C03641=1085.431,193.787,426.728,175.436,21.892,153.539
C03642=1085.437,194.036,426.705,175.438,21.893,153.539
C03643=1085.443,194.285,426.682,175.441,21.895,153.539
C03644=1085.448,194.534,426.658,175.443,21.897,153.539
C03645=1085.453,194.783,426.636,175.446,21.899,153.539
C03646=1085.459,195.032,426.613,175.448,21.900,153.539
C03647=1085.465,195.280,426.589,175.451,21.902,153.539
C03648=1085.470,195.530,426.565,175.453,21.904,153.539
C03649=1085.476,195.779,426.542,175.457,21.906,153.539
C03650=1085.482,196.027,426.519,175.459,21.907,153.539
C03651=1085.487,196.277,426.496,175.461,21.909,153.539
C03652=1085.493,196.525,426.472,175.464,21.911,153.539
C03653=1085.498,196.774,426.449,175.467,21.912,153.539
C03654=1085.504,197.023,426.426,175.469,21.914,153.539
C03655=1085.510,197.271,426.402,175.471,21.916,153.539
C03656=1085.515,197.520,426.379,175.474,21.917,153.539
C03657=1085.521,197.769,426.356,175.476,21.919,153.539
C03658=1085.526,198.018,426.333,175.479,21.921,153.539
C03659=1085.532,198.267,426.309,175.482,21.923,153.539
C03660=1085.538,198.515,426.286,175.485,21.925,153.539
C03661=1085.543,198.765,426.263,175.487,21.927,153.539
C03662=1085.549,199.013,426.239,175.490,21.928,153.539
C03663=1085.554,199.262,426.216,175.492,21.930,153.539
C03664=1085.560,199.510,426.192,175.495,21.932,153.539
C03665=1085.566,199.759,426.169,175.497,21.933,153.539
C03666=1085.572,200.009,426.145,175.500,21.935,153.539
C03667=1085.577,200.258,426.121,175.502,21.937,153.539
C03668=1085.583,200.506,426.098,175.505,21.938,153.539
C03669=1085.589,200.755,426.075,175.508,21.940,153.539
C03670=1085.594,201.004,426.051,175.511,21.942,153.538
C03671=1085.600,201.252,426.027,175.513,21.944,153.539
C03672=1085.605,201.501,426.004,175.516,21.945,153.539
C03673=1085.612,201.750,425.980,175.518,21.947,153.538
C03674=1085.617,201.999,425.957,175.521,21.949,153.538
C03675=1085.623,202.248,425.933,175.523,21.950,153.538
C03676=1085.628,202.497,425.910,175.526,21.952,153.538
C03677=1085.634,202.745,425.885,175.529,21.954,153.538
C03678=1085.639,202.994,425.862,175.532,21.956,153.538
C03679=1085.645,203.243,425.838,175.534,21.957,153.538
C03680=1085.651,203.492,425.815,175.537,21.959,153.538
C03681=1085.656,203.741,425.791,175.539,21.961,153.538
C03682=1085.661,203.990,425.767,175.542,21.963,153.538
C03683=1085.667,204.239,425.743,175.544,21.964,153.538
C03684=1085.673,204.487,425.719,175.548,21.966,153.538
C03685=1085.678,204.736,425.696,175.550,21.968,153.538
C03686=1085.684,204.985,425.672,175.553,21.970,153.538
C03687=1085.689,205.233,425.648,175.555,21.972,153.538
C03688=1085.695,205.483,425.624,175.558,21.973,153.538
C03689=1085.701,205.731,425.600,175.560,21.975,153.538
C03690=1085.706,205.980,425.576,175.564,21.977,153.538
C03691=1085.712,206.229,425.553,175.566,21.979,153.538
C03692=1085.717,206.477,425.529,175.568,21.981,153.538
C03693=1085.724,206.726,425.505,175.571,21.983,153.538
C03694=1085.729,206.976,425.481,175.574,21.984,153.538
C03695=1085.734,207.224,425.457,175.576,21.986,153.538
C03696=1085.757,208.251,425.358,175.658,22.028,153.535
C03697=1085.767,208.639,425.320,175.662,22.033,153.535
C03698=1085.775,209.027,425.282,175.666,22.037,153.535
C03699=1085.783,209.415,425.244,175.670,22.041,153.536
C03700=1085.793,209.803,425.205,175.673,22.045,153.536
C03701=1085.798,210.051,425.181,175.676,22.048,153.536
C03702=1085.804,210.301,425.157,175.678,22.050,153.536
C03703=1085.810,210.549,425.132,175.681,22.053,153.536
C03704=1085.815,210.798,425.108,175.684,22.056,153.537
C03705=1085.821,211.047,425.083,175.686,22.058,153.537
C03706=1085.826,211.295,425.058,175.689,22.061,153.537
C03707=1085.832,211.544,425.034,175.691,22.064,153.537
C03708=1085.838,211.793,425.010,175.694,22.067,153.538
C03709=1085.843,212.042,424.985,175.696,22.069,153.538
C03710=1085.849,212.290,424.960,175.699,22.072,153.538
C03711=1085.854,212.539,424.936,175.701,22.075,153.538
C03712=1085.860,212.788,424.911,175.704,22.077,153.538
C03713=1085.866,213.036,424.886,175.707,22.080,153.538
C03714=1085.872,213.285,424.862,175.709,22.083,153.539
C03715=1085.877,213.534,424.837,175.712,22.086,153.539
C03716=1085.882,213.784,424.812,175.714,22.088,153.539
C03717=1085.888,214.032,424.787,175.716,22.091,153.539
C03718=1085.894,214.281,424.762,175.720,22.094,153.539
C03719=1085.899,214.529,424.737,175.722,22.096,153.540
C03720=1085.905,214.777,424.713,175.725,22.099,153.540
C03721=1085.910,215.027,424.689,175.727,22.102,153.540
C03722=1085.916,215.275,424.664,175.730,22.105,153.540
C03723=1085.921,215.524,424.638,175.732,22.107,153.540
C03724=1085.927,215.772,424.613,175.734,22.110,153.541
C03725=1085.933,216.022,424.589,175.737,22.113,153.541
C03726=1085.938,216.270,424.564,175.740,22.115,153.541
C03727=1085.944,216.519,424.539,175.743,22.118,153.541
C03728=1085.949,216.767,424.514,175.745,22.121,153.541
C03729=1085.955,217.016,424.489,175.748,22.124,153.542
C03730=1085.961,217.264,424.464,175.750,22.126,153.542
C03731=1085.967,217.514,424.439,175.753,22.129,153.542
C03732=1085.973,217.762,424.414,175.755,22.132,153.542
C03733=1085.977,218.011,424.389,175.757,22.134,153.542
C03734=1085.984,218.260,424.364,175.761,22.137,153.543
C03735=1085.989,218.508,424.340,175.763,22.139,153.543
C03736=1085.995,218.757,424.314,175.766,22.143,153.543
C03737=1086.000,219.006,424.290,175.768,22.145,153.543
C03738=1086.006,219.255,424.264,175.771,22.148,153.543
C03739=1086.012,219.503,424.239,175.773,22.151,153.544
C03740=1086.017,219.752,424.215,175.776,22.153,153.544
C03741=1086.023,220.001,424.189,175.779,22.156,153.544
C03742=1086.028,220.249,424.164,175.782,22.159,153.544
C03743=1086.034,220.498,424.139,175.784,22.161,153.544
C03744=1086.040,220.747,424.114,175.786,22.164,153.544
C03745=1086.046,220.995,424.089,175.789,22.167,153.545
C03746=1086.051,221.244,424.063,175.791,22.169,153.545
C03747=1086.057,221.493,424.038,175.794,22.172,153.545
C03748=1086.063,221.741,424.013,175.797,22.175,153.545
C03749=1086.072,222.133,423.973,175.801,22.179,153.546
C03750=1086.081,222.526,423.934,175.805,22.183,153.546
C03751=1086.090,222.917,423.893,175.809,22.188,153.546
C03752=1086.098,223.309,423.854,175.813,22.192,153.547
C03753=1086.103,223.558,423.828,175.816,22.195,153.547
C03754=1086.109,223.806,423.803,175.818,22.197,153.547
C03755=1086.115,224.054,423.778,175.821,22.201,153.547
C03756=1086.121,224.303,423.752,175.824,22.203,153.547
C03757=1086.126,224.553,423.727,175.827,22.206,153.548
C03758=1086.131,224.801,423.702,175.829,22.209,153.548
C03759=1086.138,225.050,423.676,175.832,22.211,153.548
C03760=1086.143,225.298,423.650,175.834,22.214,153.548
C03761=1086.149,225.546,423.625,175.837,22.217,153.548
C03762=1086.154,225.795,423.599,175.839,22.219,153.548
C03763=1086.160,226.044,423.574,175.842,22.223,153.549
C03764=1086.165,226.292,423.548,175.845,22.225,153.549
C03765=1086.171,226.541,423.523,175.848,22.228,153.549
C03766=1086.177,226.790,423.497,175.850,22.231,153.549
C03767=1086.182,227.039,423.471,175.853,22.233,153.549
C03768=1086.188,227.287,423.446,175.855,22.236,153.550
C03769=1086.193,227.536,423.420,175.858,22.239,153.550
C03770=1086.200,227.785,423.395,175.860,22.241,153.550
C03771=1086.205,228.034,423.369,175.863,22.245,153.550
C03772=1086.211,228.282,423.344,175.866,22.247,153.551
C03773=1086.216,228.531,423.318,175.869,22.250,153.551
C03774=1086.222,228.779,423.293,175.871,22.252,153.551
C03775=1086.228,229.028,423.267,175.874,22.255,153.551
C03776=1086.234,229.277,423.240,175.876,22.258,153.551
C03777=1086.239,229.525,423.215,175.879,22.261,153.552
C03778=1086.245,229.774,423.189,175.881,22.263,153.552
C03779=1086.251,230.022,423.164,175.885,22.266,153.552
C03780=1086.256,230.271,423.138,175.887,22.269,153.552
C03781=1086.262,230.520,423.112,175.890,22.272,153.552
C03782=1086.267,230.768,423.087,175.892,22.274,153.552
C03783=1086.273,231.016,423.061,175.895,22.277,153.553
C03784=1086.279,231.265,423.035,175.898,22.280,153.553
C03785=1086.284,231.514,423.009,175.900,22.283,153.553
C03786=1086.290,231.763,422.983,175.903,22.285,153.553
C03787=1086.295,232.011,422.957,175.905,22.288,153.554
C03788=1086.301,232.260,422.931,175.909,22.291,153.554
C03789=1086.306,232.509,422.905,175.911,22.293,153.554
C03790=1086.313,232.757,422.880,175.914,22.297,153.554
C03791=1086.318,233.006,422.853,175.916,22.299,153.554
C03792=1086.324,233.255,422.827,175.919,22.302,153.555
C03793=1086.329,233.503,422.802,175.921,22.305,153.555
C03794=1086.335,233.751,422.776,175.924,22.307,153.555
C03795=1086.341,234.000,422.750,175.927,22.310,153.555
C03796=1086.346,234.248,422.723,175.930,22.313,153.555
C03797=1086.352,234.497,422.697,175.933,22.316,153.556
C03798=1086.357,234.746,422.671,175.935,22.319,153.556
C03799=1086.363,234.995,422.645,175.938,22.322,153.556
C03800=1086.368,235.243,422.619,175.940,22.324,153.556
C03801=1086.377,235.626,422.579,175.945,22.329,153.556
C03802=1086.386,236.010,422.538,175.948,22.333,153.557
C03803=1086.394,236.393,422.498,175.953,22.337,153.557
C03804=1086.404,236.777,422.458,175.957,22.341,153.557
C03805=1086.409,237.025,422.431,175.960,22.344,153.558
C03806=1086.414,237.273,422.405,175.962,22.347,153.558
C03807=1086.420,237.522,422.379,175.965,22.350,153.558
C03808=1086.425,237.771,422.353,175.968,22.353,153.558
C03809=1086.431,238.019,422.326,175.970,22.355,153.558
C03810=1086.437,238.267,422.300,175.973,22.359,153.559
C03811=1086.442,238.516,422.274,175.976,22.361,153.559
C03812=1086.448,238.765,422.247,175.979,22.364,153.559
C03813=1086.454,239.014,422.221,175.981,22.366,153.559
C03814=1086.459,239.262,422.194,175.984,22.369,153.559
C03815=1086.465,239.510,422.168,175.987,22.372,153.560
C03816=1086.471,239.759,422.142,175.989,22.375,153.560
C03817=1086.476,240.008,422.115,175.992,22.378,153.560
C03818=1086.482,240.256,422.088,175.994,22.380,153.560
C03819=1086.488,240.505,422.063,175.998,22.383,153.560
C03820=1086.493,240.753,422.036,176.001,22.386,153.561
C03821=1086.499,241.002,422.009,176.003,22.389,153.561
C03822=1086.505,241.250,421.983,176.006,22.391,153.561
C03823=1086.510,241.499,421.957,176.008,22.394,153.561
C03824=1086.516,241.747,421.930,176.011,22.397,153.561
C03825=1086.522,241.996,421.903,176.014,22.400,153.562
C03826=1086.528,242.244,421.877,176.016,22.403,153.562
C03827=1086.533,242.493,421.851,176.019,22.406,153.562
C03828=1086.539,242.742,421.824,176.022,22.408,153.562
C03829=1086.545,242.990,421.798,176.025,22.411,153.563
C03830=1086.551,243.238,421.771,176.028,22.414,153.563
C03831=1086.556,243.488,421.743,176.030,22.417,153.563
C03832=1086.562,243.736,421.717,176.033,22.420,153.563
C03833=1086.568,243.984,421.690,176.035,22.422,153.563
C03834=1086.573,244.233,421.664,176.038,22.425,153.564
C03835=1086.579,244.482,421.637,176.041,22.428,153.564
C03836=1086.584,244.730,421.610,176.043,22.431,153.564
C03837=1086.590,244.979,421.583,176.047,22.434,153.564
C03838=1086.596,245.227,421.557,176.050,22.437,153.565
C03839=1086.601,245.475,421.530,176.052,22.439,153.565
C03840=1086.606,245.724,421.503,176.055,22.443,153.565
C03841=1086.612,245.972,421.476,176.057,22.445,153.565
C03842=1086.618,246.221,421.450,176.060,22.448,153.565
C03843=1086.623,246.470,421.422,176.063,22.451,153.566
C03844=1086.629,246.718,421.396,176.065,22.454,153.566
C03845=1086.635,246.967,421.369,176.069,22.456,153.566
C03846=1086.641,247.215,421.342,176.071,22.460,153.566
C03847=1086.646,247.464,421.315,176.074,22.462,153.566
C03848=1086.652,247.712,421.288,176.077,22.465,153.567
C03849=1086.657,247.961,421.261,176.080,22.468,153.567
C03850=1086.663,248.209,421.234,176.082,22.471,153.567
C03851=1086.668,248.457,421.206,176.085,22.474,153.567
C03852=1086.674,248.706,421.180,176.087,22.476,153.568
C03853=1086.682,249.083,421.139,176.092,22.481,153.568
C03854=1086.690,249.459,421.098,176.096,22.486,153.568
C03855=1086.699,249.835,421.057,176.100,22.490,153.569
C03856=1086.707,250.211,421.016,176.105,22.494,153.569
C03857=1086.712,250.460,420.988,176.107,22.497,153.569
C03858=1086.719,250.709,420.961,176.110,22.500,153.569
C03859=1086.724,250.957,420.933,176.113,22.503,153.570
C03860=1086.730,251.206,420.907,176.115,22.506,153.570
C03861=1086.735,251.454,420.880,176.118,22.509,153.570
C03862=1086.741,251.703,420.853,176.121,22.512,153.570
C03863=1086.746,251.951,420.825,176.123,22.514,153.571
C03864=1086.752,252.200,420.798,176.126,22.518,153.571
C03865=1086.758,252.448,420.771,176.129,22.520,153.571
C03866=1086.764,252.696,420.743,176.132,22.523,153.571
C03867=1086.769,252.945,420.716,176.135,22.526,153.571
C03868=1086.774,253.193,420.689,176.138,22.529,153.572
C03869=1086.780,253.442,420.661,176.140,22.532,153.572
C03870=1086.785,253.691,420.634,176.143,22.535,153.572
C03871=1086.791,253.938,420.607,176.146,22.538,153.572
C03872=1086.796,254.187,420.579,176.148,22.540,153.573
C03873=1086.803,254.435,420.552,176.151,22.543,153.573
C03874=1086.808,254.684,420.524,176.154,22.546,153.573
C03875=1086.814,254.932,420.496,176.156,22.549,153.573
C03876=1086.820,255.181,420.469,176.160,22.552,153.574
C03877=1086.825,255.430,420.442,176.163,22.555,153.574
C03878=1086.831,255.678,420.415,176.165,22.558,153.574
C03879=1086.836,255.926,420.387,176.168,22.561,153.574
C03880=1086.842,256.175,420.359,176.171,22.564,153.575
C03881=1086.848,256.423,420.332,176.174,22.567,153.575
C03882=1086.853,256.671,420.305,176.176,22.569,153.575
C03883=1086.860,256.920,420.277,176.179,22.572,153.575
C03884=1086.865,257.169,420.250,176.182,22.575,153.575
C03885=1086.870,257.417,420.222,176.184,22.578,153.576
C03886=1086.877,257.665,420.194,176.187,22.581,153.576
C03887=1086.882,257.914,420.167,176.190,22.584,153.576
C03888=1086.887,258.162,420.139,176.193,22.586,153.576
C03889=1086.894,258.410,420.111,176.196,22.590,153.577
C03890=1086.899,258.659,420.084,176.199,22.592,153.577
C03891=1086.905,258.908,420.055,176.202,22.596,153.577
C03892=1086.911,259.155,420.028,176.204,22.598,153.577
C03893=1086.916,259.404,420.001,176.207,22.601,153.577
C03894=1086.922,259.653,419.972,176.210,22.604,153.578
C03895=1086.928,259.900,419.945,176.212,22.607,153.578
C03896=1086.934,260.149,419.917,176.216,22.609,153.578
C03897=1086.939,260.398,419.890,176.219,22.613,153.578
C03898=1086.945,260.646,419.862,176.222,22.616,153.579
C03899=1086.951,260.894,419.834,176.224,22.618,153.579
C03900=1086.956,261.142,419.806,176.227,22.621,153.579
C03901=1086.963,261.391,419.778,176.230,22.624,153.579
C03902=1086.968,261.640,419.751,176.233,22.627,153.579
C03903=1086.974,261.888,419.723,176.235,22.630,153.580
C03904=1086.979,262.136,419.695,176.238,22.633,153.580
C03905=1086.989,262.510,419.653,176.243,22.638,153.580
C03906=1086.997,262.883,419.610,176.247,22.641,153.581
C03907=1087.006,263.257,419.569,176.251,22.646,153.581
C03908=1087.014,263.630,419.526,176.256,22.650,153.581
C03909=1087.021,263.879,419.499,176.258,22.653,153.581
C03910=1087.026,264.127,419.471,176.261,22.656,153.582
C03911=1087.032,264.376,419.443,176.264,22.659,153.582
C03912=1087.037,264.624,419.415,176.266,22.662,153.582
C03913=1087.043,264.873,419.387,176.269,22.665,153.582
C03914=1087.049,265.120,419.358,176.272,22.668,153.583
C03915=1087.055,265.369,419.330,176.276,22.671,153.583
C03916=1087.060,265.617,419.302,176.279,22.674,153.583
C03917=1087.066,265.866,419.273,176.281,22.677,153.583
C03918=1087.072,266.114,419.245,176.284,22.680,153.584
C03919=1087.078,266.363,419.217,176.287,22.683,153.584
C03920=1087.083,266.611,419.189,176.290,22.686,153.584
C03921=1087.089,266.859,419.161,176.292,22.689,153.584
C03922=1087.094,267.107,419.133,176.295,22.691,153.585
C03923=1087.100,267.356,419.104,176.298,22.695,153.585
C03924=1087.106,267.604,419.076,176.301,22.698,153.585
C03925=1087.112,267.852,419.047,176.303,22.700,153.585
C03926=1087.117,268.100,419.019,176.306,22.703,153.586
C03927=1087.123,268.349,418.991,176.309,22.707,153.586
C03928=1087.129,268.598,418.963,176.312,22.710,153.586
C03929=1087.135,268.845,418.934,176.315,22.713,153.586
C03930=1087.141,269.094,418.906,176.318,22.715,153.587
C03931=1087.145,269.343,418.877,176.321,22.719,153.587
C03932=1087.151,269.591,418.848,176.324,22.721,153.587
C03933=1087.157,269.839,418.820,176.327,22.725,153.587
C03934=1087.163,270.087,418.792,176.329,22.727,153.588
C03935=1087.169,270.336,418.764,176.332,22.731,153.588
C03936=1087.174,270.584,418.735,176.335,22.733,153.588
C03937=1087.180,270.832,418.707,176.338,22.737,153.588
C03938=1087.185,271.080,418.677,176.341,22.740,153.589
C03939=1087.191,271.329,418.649,176.343,22.743,153.589
C03940=1087.197,271.578,418.621,176.346,22.745,153.589
C03941=1087.203,271.825,418.592,176.349,22.749,153.589
C03942=1087.209,272.074,418.564,176.352,22.752,153.590
C03943=1087.214,272.322,418.534,176.355,22.755,153.590
C03944=1087.219,272.570,418.506,176.357,22.758,153.590
C03945=1087.226,272.818,418.477,176.361,22.760,153.590
C03946=1087.231,273.066,418.449,176.364,22.764,153.591
C03947=1087.237,273.315,418.419,176.367,22.767,153.591
C03948=1087.242,273.564,418.391,176.370,22.770,153.591
C03949=1087.248,273.811,418.362,176.372,22.772,153.591
C03950=1087.254,274.060,418.334,176.375,22.776,153.592
C03951=1087.260,274.308,418.304,176.378,22.779,153.592
C03952=1087.265,274.556,418.277,176.381,22.782,153.592
C03953=1087.270,274.805,418.247,176.384,22.785,153.593
C03954=1087.276,275.054,418.219,176.387,22.789,153.593
C03955=1087.282,275.301,418.190,176.389,22.791,153.593
C03956=1087.288,275.549,418.160,176.392,22.794,153.593
C03957=1087.296,275.926,418.117,176.397,22.799,153.594
C03958=1087.304,276.302,418.073,176.401,22.804,153.594
C03959=1087.313,276.678,418.030,176.406,22.808,153.594
C03960=1087.322,277.055,417.985,176.409,22.813,153.595
C03961=1087.328,277.303,417.956,176.412,22.816,153.595
C03962=1087.333,277.552,417.927,176.415,22.819,153.596
C03963=1087.339,277.800,417.898,176.419,22.822,153.596
C03964=1087.345,278.049,417.869,176.422,22.825,153.596
C03965=1087.351,278.296,417.840,176.425,22.828,153.596
C03966=1087.356,278.544,417.810,176.427,22.831,153.597
C03967=1087.362,278.793,417.782,176.430,22.834,153.597
C03968=1087.368,279.042,417.753,176.433,22.838,153.597
C03969=1087.373,279.289,417.724,176.436,22.841,153.597
C03970=1087.379,279.537,417.694,176.439,22.844,153.598
C03971=1087.385,279.786,417.665,176.442,22.847,153.598
C03972=1087.390,280.034,417.636,176.445,22.851,153.598
C03973=1087.396,280.281,417.607,176.447,22.853,153.598
C03974=1087.402,280.530,417.577,176.450,22.856,153.599
C03975=1087.408,280.779,417.549,176.453,22.859,153.599
C03976=1087.413,281.027,417.519,176.456,22.862,153.599
C03977=1087.419,281.275,417.490,176.459,22.866,153.600
C03978=1087.424,281.523,417.461,176.462,22.869,153.600
C03979=1087.431,281.771,417.432,176.465,22.872,153.600
C03980=1087.436,282.020,417.402,176.467,22.875,153.601
C03981=1087.442,282.268,417.373,176.470,22.878,153.601
C03982=1087.448,282.516,417.344,176.473,22.881,153.601
C03983=1087.453,282.764,417.314,176.476,22.884,153.601
C03984=1087.458,283.012,417.285,176.479,22.888,153.602
C03985=1087.464,283.260,417.254,176.482,22.891,153.602
C03986=1087.470,283.508,417.225,176.485,22.894,153.602
C03987=1087.476,283.757,417.196,176.488,22.897,153.603
C03988=1087.481,284.005,417.166,176.491,22.900,153.603
C03989=1087.487,284.253,417.137,176.493,22.903,153.603
C03990=1087.492,284.501,417.108,176.496,22.907,153.604
C03991=1087.498,284.749,417.078,176.499,22.910,153.604
C03992=1087.503,284.998,417.048,176.502,22.913,153.604
C03993=1087.510,285.245,417.019,176.505,22.917,153.604
C03994=1087.516,285.494,416.989,176.508,22.920,153.605
C03995=1087.521,285.742,416.959,176.511,22.923,153.605
C03996=1087.527,285.990,416.930,176.514,22.926,153.605
C03997=1087.533,286.238,416.900,176.517,22.929,153.606
C03998=1087.538,286.486,416.871,176.519,22.932,153.606
C03999=1087.544,286.734,416.841,176.522,22.935,153.606
C04000=1087.549,286.983,416.812,176.525,22.939,153.606
C04001=1087.556,287.230,416.782,176.528,22.942,153.607
C04002=1087.561,287.479,416.752,176.531,22.945,153.607
C04003=1087.567,287.727,416.722,176.534,22.948,153.607
C04004=1087.572,287.975,416.692,176.537,22.951,153.608
C04005=1087.579,288.223,416.663,176.540,22.955,153.608
C04006=1087.584,288.472,416.633,176.544,22.958,153.608
C04007=1087.590,288.719,416.603,176.547,22.961,153.608
C04008=1087.596,288.968,416.573,176.549,22.965,153.609
C04009=1087.604,289.354,416.527,176.554,22.969,153.609
C04010=1087.613,289.740,416.480,176.558,22.974,153.610
C04011=1087.622,290.125,416.434,176.563,22.979,153.610
C04012=1087.631,290.511,416.387,176.567,22.984,153.611
C04013=1087.636,290.760,416.357,176.570,22.988,153.611
C04014=1087.642,291.007,416.327,176.573,22.991,153.611
C04015=1087.648,291.256,416.297,176.576,22.994,153.612
C04016=1087.654,291.504,416.267,176.579,22.998,153.612
C04017=1087.660,291.752,416.238,176.582,23.001,153.612
C04018=1087.666,292.000,416.208,176.585,23.004,153.613
C04019=1087.671,292.248,416.178,176.588,23.007,153.613
C04020=1087.677,292.496,416.148,176.591,23.011,153.613
C04021=1087.682,292.744,416.117,176.594,23.014,153.614
C04022=1087.688,292.992,416.087,176.597,23.017,153.614
C04023=1087.694,293.241,416.056,176.599,23.020,153.614
C04024=1087.700,293.489,416.026,176.602,23.024,153.615
C04025=1087.705,293.737,415.996,176.605,23.027,153.615
C04026=1087.711,293.985,415.966,176.608,23.030,153.615
C04027=1087.717,294.233,415.936,176.611,23.033,153.615
C04028=1087.723,294.481,415.905,176.614,23.037,153.616
C04029=1087.728,294.729,415.876,176.617,23.040,153.616
C04030=1087.734,294.977,415.845,176.620,23.043,153.616
C04031=1087.740,295.225,415.815,176.623,23.046,153.617
C04032=1087.746,295.473,415.785,176.626,23.050,153.617
C04033=1087.751,295.721,415.755,176.629,23.053,153.617
C04034=1087.757,295.969,415.725,176.632,23.057,153.618
C04035=1087.763,296.218,415.693,176.635,23.060,153.618
C04036=1087.769,296.466,415.663,176.638,23.063,153.618
C04037=1087.774,296.713,415.633,176.641,23.067,153.619
C04038=1087.780,296.961,415.602,176.644,23.070,153.619
C04039=1087.786,297.209,415.572,176.647,23.073,153.619
C04040=1087.791,297.458,415.542,176.650,23.077,153.620
C04041=1087.797,297.706,415.511,176.653,23.080,153.620
C04042=1087.803,297.954,415.481,176.656,23.084,153.620
C04043=1087.809,298.202,415.450,176.659,23.087,153.621
C04044=1087.814,298.450,415.419,176.662,23.090,153.621
C04045=1087.820,298.698,415.389,176.665,23.094,153.621
C04046=1087.825,298.946,415.358,176.667,23.097,153.622
C04047=1087.831,299.194,415.328,176.670,23.101,153.622
C04048=1087.837,299.442,415.297,176.673,23.104,153.623
C04049=1087.842,299.690,415.266,176.676,23.108,153.623
C04050=1087.847,299.938,415.236,176.679,23.111,153.623
C04051=1087.853,300.186,415.204,176.682,23.115,153.624
C04052=1087.859,300.434,415.174,176.685,23.118,153.624
C04053=1087.864,300.682,415.143,176.688,23.121,153.624
C04054=1087.870,300.930,415.112,176.691,23.125,153.625
C04055=1087.876,301.177,415.082,176.694,23.128,153.625
C04056=1087.881,301.426,415.051,176.697,23.132,153.626
C04057=1087.887,301.674,415.020,176.700,23.135,153.626
C04058=1087.893,301.922,414.989,176.703,23.139,153.626
C04059=1087.899,302.169,414.958,176.706,23.142,153.627
C04060=1087.904,302.418,414.927,176.708,23.146,153.627
C04061=1087.913,302.818,414.878,176.714,23.152,153.628
C04062=1087.922,303.217,414.828,176.718,23.157,153.628
C04063=1087.932,303.618,414.778,176.723,23.163,153.629
C04064=1087.940,304.018,414.728,176.728,23.168,153.629
C04065=1087.946,304.265,414.697,176.731,23.172,153.630
C04066=1087.952,304.514,414.665,176.734,23.175,153.630
C04067=1087.958,304.762,414.635,176.737,23.179,153.631
C04068=1087.963,305.010,414.604,176.740,23.183,153.631
C04069=1087.969,305.257,414.573,176.743,23.186,153.631
C04070=1087.975,305.506,414.542,176.746,23.189,153.632
C04071=1087.981,305.753,414.511,176.749,23.193,153.632
C04072=1087.986,306.001,414.480,176.752,23.196,153.632
C04073=1087.992,306.250,414.448,176.755,23.200,153.633
C04074=1087.998,306.497,414.417,176.758,23.203,153.633
C04075=1088.003,306.745,414.386,176.761,23.207,153.634
C04076=1088.010,306.993,414.355,176.764,23.210,153.634
C04077=1088.015,307.241,414.324,176.767,23.214,153.634
C04078=1088.021,307.488,414.293,176.769,23.217,153.635
C04079=1088.026,307.737,414.262,176.773,23.221,153.635
C04080=1088.032,307.985,414.230,176.776,23.224,153.635
C04081=1088.039,308.233,414.198,176.779,23.228,153.636
C04082=1088.044,308.481,414.168,176.782,23.232,153.636
C04083=1088.050,308.728,414.136,176.785,23.235,153.637
C04084=1088.055,308.977,414.105,176.788,23.239,153.637
C04085=1088.061,309.224,414.073,176.791,23.242,153.637
C04086=1088.068,309.472,414.042,176.794,23.246,153.638
C04087=1088.073,309.720,414.011,176.797,23.249,153.638
C04088=1088.078,309.968,413.979,176.800,23.253,153.639
C04089=1088.085,310.216,413.948,176.802,23.256,153.639
C04090=1088.090,310.464,413.917,176.806,23.260,153.639
C04091=1088.096,310.712,413.885,176.809,23.264,153.640
C04092=1088.102,310.959,413.854,176.812,23.267,153.640
C04093=1088.108,311.208,413.823,176.815,23.271,153.641
C04094=1088.113,311.456,413.791,176.818,23.274,153.641
C04095=1088.120,311.704,413.760,176.821,23.278,153.641
C04096=1088.125,311.951,413.728,176.824,23.281,153.642
C04097=1088.131,312.199,413.696,176.827,23.285,153.642
C04098=1088.136,312.447,413.665,176.830,23.288,153.642
C04099=1088.143,312.695,413.634,176.833,23.292,153.643
C04100=1088.149,312.944,413.601,176.836,23.296,153.643
C04101=1088.154,313.191,413.570,176.839,23.300,153.644
C04102=1088.161,313.439,413.538,176.842,23.303,153.644
C04103=1088.166,313.686,413.507,176.845,23.306,153.644
C04104=1088.172,313.935,413.475,176.848,23.310,153.645
C04105=1088.177,314.183,413.444,176.851,23.314,153.645
C04106=1088.184,314.431,413.412,176.854,23.317,153.646
C04107=1088.190,314.679,413.380,176.857,23.321,153.646
C04108=1088.196,314.926,413.349,176.861,23.325,153.646
C04109=1088.201,315.175,413.317,176.863,23.328,153.647
C04110=1088.207,315.422,413.285,176.866,23.332,153.647
C04111=1088.213,315.670,413.253,176.869,23.336,153.648
C04112=1088.218,315.918,413.221,176.872,23.340,153.648
C04113=1088.225,316.226,413.181,176.875,23.344,153.649
C04114=1088.232,316.532,413.141,176.879,23.349,153.649
C04115=1088.239,316.841,413.102,176.884,23.354,153.650
C04116=1088.246,317.147,413.062,176.887,23.359,153.651
C04117=1088.252,317.395,413.030,176.890,23.362,153.651
C04118=1088.258,317.643,412.999,176.893,23.366,153.651
C04119=1088.263,317.891,412.966,176.896,23.370,153.652
C04120=1088.269,318.138,412.934,176.899,23.373,153.652
C04121=1088.275,318.387,412.902,176.901,23.377,153.653
C04122=1088.281,318.635,412.870,176.905,23.381,153.653
C04123=1088.286,318.882,412.838,176.908,23.385,153.654
C04124=1088.292,319.130,412.806,176.911,23.389,153.654
C04125=1088.297,319.378,412.773,176.914,23.392,153.654
C04126=1088.303,319.626,412.741,176.916,23.396,153.655
C04127=1088.309,319.874,412.709,176.919,23.400,153.655
C04128=1088.314,320.122,412.677,176.923,23.404,153.656
C04129=1088.321,320.369,412.644,176.926,23.408,153.656
C04130=1088.326,320.618,412.612,176.929,23.412,153.657
C04131=1088.331,320.865,412.580,176.932,23.415,153.657
C04132=1088.337,321.113,412.547,176.934,23.419,153.658
C04133=1088.343,321.361,412.515,176.938,23.424,153.658
C04134=1088.348,321.609,412.483,176.941,23.427,153.659
C04135=1088.354,321.856,412.450,176.944,23.431,153.659
C04136=1088.360,322.105,412.418,176.947,23.435,153.660
C04137=1088.366,322.352,412.386,176.949,23.439,153.660
C04138=1088.371,322.600,412.353,176.953,23.443,153.661
C04139=1088.378,322.848,412.321,176.956,23.447,153.661
C04140=1088.384,323.096,412.289,176.959,23.450,153.662
C04141=1088.391,323.439,412.244,176.963,23.456,153.662
C04142=1088.399,323.783,412.199,176.967,23.461,153.663
C04143=1088.408,324.126,412.153,176.971,23.466,153.664
C04144=1088.415,324.469,412.109,176.975,23.472,153.664
C04145=1088.421,324.717,412.075,176.979,23.476,153.665
C04146=1088.427,324.965,412.043,176.982,23.480,153.665
C04147=1088.433,325.212,412.011,176.985,23.484,153.666
C04148=1088.438,325.460,411.978,176.987,23.488,153.666
C04149=1088.444,325.708,411.946,176.990,23.491,153.667
C04150=1088.450,325.955,411.913,176.994,23.496,153.667
C04151=1088.456,326.204,411.880,176.997,23.499,153.668
C04152=1088.462,326.452,411.848,177.000,23.504,153.668
C04153=1088.468,326.699,411.815,177.002,23.507,153.669
C04154=1088.473,326.948,411.782,177.006,23.512,153.669
C04155=1088.479,327.195,411.750,177.009,23.515,153.670
C04156=1088.485,327.442,411.717,177.012,23.519,153.670
C04157=1088.491,327.690,411.684,177.015,23.523,153.671
C04158=1088.497,327.938,411.652,177.018,23.528,153.671
C04159=1088.502,328.186,411.618,177.021,23.531,153.672
C04160=1088.509,328.434,411.586,177.024,23.535,153.672
C04161=1088.515,328.681,411.553,177.027,23.539,153.673
C04162=1088.521,328.929,411.520,177.030,23.543,153.673
C04163=1088.527,329.177,411.487,177.033,23.547,153.673
C04164=1088.532,329.425,411.454,177.036,23.551,153.674
C04165=1088.542,329.821,411.402,177.041,23.557,153.675
C04166=1088.551,330.217,411.350,177.046,23.564,153.676
C04167=1088.561,330.613,411.296,177.051,23.571,153.676
C04168=1088.570,331.009,411.243,177.056,23.577,153.677
C04169=1088.577,331.256,411.211,177.059,23.581,153.678
C04170=1088.582,331.504,411.177,177.062,23.585,153.678
C04171=1088.588,331.752,411.145,177.065,23.589,153.679
C04172=1088.594,332.000,411.111,177.068,23.593,153.679
C04173=1088.600,332.248,411.078,177.071,23.597,153.680
C04174=1088.606,332.495,411.045,177.074,23.601,153.680
C04175=1088.611,332.743,411.012,177.077,23.605,153.681
C04176=1088.617,332.991,410.979,177.080,23.609,153.681
C04177=1088.623,333.239,410.945,177.083,23.614,153.682
C04178=1088.629,333.486,410.912,177.087,23.618,153.683
C04179=1088.635,333.734,410.878,177.089,23.622,153.683
C04180=1088.640,333.982,410.845,177.092,23.626,153.684
C04181=1088.646,334.230,410.812,177.096,23.631,153.684
C04182=1088.652,334.477,410.779,177.098,23.635,153.685
C04183=1088.658,334.725,410.746,177.101,23.639,153.685
C04184=1088.664,334.972,410.712,177.105,23.643,153.686
C04185=1088.669,335.220,410.678,177.108,23.647,153.687
C04186=1088.675,335.468,410.645,177.110,23.652,153.687
C04187=1088.681,335.716,410.612,177.114,23.656,153.688
C04188=1088.687,335.963,410.578,177.117,23.660,153.688
C04189=1088.692,336.211,410.545,177.119,23.664,153.689
C04190=1088.698,336.459,410.511,177.123,23.669,153.689
C04191=1088.704,336.706,410.477,177.126,23.673,153.690
C04192=1088.711,336.954,410.444,177.129,23.677,153.690
C04193=1088.716,337.202,410.411,177.132,23.681,153.691
C04194=1088.722,337.450,410.377,177.135,23.685,153.692
C04195=1088.728,337.697,410.344,177.139,23.690,153.692
C04196=1088.733,337.945,410.310,177.141,23.694,153.693
C04197=1088.739,338.193,410.276,177.144,23.699,153.693
C04198=1088.745,338.441,410.243,177.148,23.703,153.694
C04199=1088.750,338.688,410.209,177.150,23.707,153.694
C04200=1088.757,338.936,410.175,177.153,23.711,153.695
C04201=1088.762,339.184,410.141,177.157,23.716,153.696
C04202=1088.768,339.432,410.108,177.159,23.720,153.696
C04203=1088.774,339.679,410.074,177.163,23.725,153.697
C04204=1088.780,339.926,410.040,177.166,23.729,153.697
C04205=1088.785,340.174,410.006,177.168,23.733,153.698
C04206=1088.791,340.421,409.972,177.172,23.738,153.699
C04207=1088.797,340.669,409.939,177.175,23.742,153.699
C04208=1088.803,340.917,409.904,177.178,23.747,153.700
C04209=1088.809,341.165,409.870,177.181,23.751,153.700
C04210=1088.815,341.412,409.837,177.184,23.755,153.701
C04211=1088.820,341.660,409.803,177.187,23.760,153.702
C04212=1088.826,341.907,409.769,177.190,23.764,153.702
C04213=1088.832,342.156,409.735,177.194,23.769,153.703
C04214=1088.838,342.403,409.701,177.196,23.773,153.704
C04215=1088.844,342.650,409.667,177.200,23.778,153.704
C04216=1088.850,342.897,409.633,177.203,23.782,153.705
C04217=1088.859,343.288,409.579,177.207,23.789,153.706
C04218=1088.868,343.679,409.526,177.212,23.797,153.707
C04219=1088.878,344.068,409.472,177.217,23.803,153.708
C04220=1088.887,344.459,409.419,177.222,23.811,153.709
C04221=1088.892,344.706,409.384,177.225,23.815,153.710
C04222=1088.899,344.954,409.350,177.228,23.820,153.710
C04223=1088.905,345.202,409.316,177.231,23.824,153.711
C04224=1088.910,345.449,409.282,177.234,23.829,153.711
C04225=1088.916,345.696,409.248,177.237,23.833,153.712
C04226=1088.922,345.944,409.213,177.241,23.838,153.713
C04227=1088.928,346.192,409.179,177.243,23.843,153.713
C04228=1088.934,346.439,409.145,177.247,23.847,153.714
C04229=1088.939,346.687,409.109,177.250,23.852,153.715
C04230=1088.945,346.935,409.075,177.253,23.856,153.715
C04231=1088.951,347.182,409.041,177.256,23.861,153.716
C04232=1088.957,347.430,409.006,177.259,23.866,153.717
C04233=1088.963,347.677,408.972,177.262,23.870,153.717
C04234=1088.969,347.925,408.938,177.265,23.875,153.718
C04235=1088.975,348.172,408.903,177.268,23.879,153.719
C04236=1088.981,348.420,408.868,177.272,23.884,153.719
C04237=1088.986,348.667,408.834,177.274,23.889,153.720
C04238=1088.992,348.915,408.799,177.278,23.894,153.721
C04239=1088.998,349.163,408.765,177.280,23.898,153.721
C04240=1089.003,349.410,408.731,177.284,23.903,153.722
C04241=1089.010,349.658,408.696,177.286,23.908,153.723
C04242=1089.016,349.905,408.662,177.290,23.913,153.724
C04243=1089.021,350.153,408.627,177.293,23.917,153.724
C04244=1089.027,350.400,408.592,177.296,23.922,153.725
C04245=1089.033,350.647,408.557,177.299,23.927,153.726
C04246=1089.039,350.895,408.523,177.302,23.932,153.726
C04247=1089.044,351.143,408.488,177.305,23.936,153.727
C04248=1089.051,351.390,408.453,177.308,23.941,153.728
C04249=1089.057,351.638,408.419,177.311,23.946,153.728
C04250=1089.062,351.885,408.383,177.315,23.951,153.729
C04251=1089.069,352.133,408.349,177.317,23.956,153.730
C04252=1089.074,352.380,408.314,177.321,23.961,153.731
C04253=1089.081,352.628,408.279,177.324,23.965,153.731
C04254=1089.086,352.875,408.245,177.327,23.970,153.732
C04255=1089.093,353.122,408.209,177.330,23.975,153.733
C04256=1089.098,353.370,408.175,177.333,23.980,153.734
C04257=1089.104,353.618,408.139,177.336,23.985,153.734
C04258=1089.110,353.865,408.105,177.339,23.989,153.735
C04259=1089.116,354.113,408.069,177.342,23.995,153.736
C04260=1089.122,354.360,408.035,177.345,23.999,153.736
C04261=1089.128,354.608,408.000,177.348,24.004,153.737
C04262=1089.133,354.855,407.964,177.352,24.010,153.738
C04263=1089.139,355.103,407.930,177.354,24.014,153.739
C04264=1089.145,355.350,407.894,177.358,24.019,153.739
C04265=1089.151,355.598,407.859,177.360,24.024,153.740
C04266=1089.156,355.845,407.824,177.364,24.029,153.741
C04267=1089.163,356.092,407.789,177.367,24.034,153.742
C04268=1089.168,356.339,407.754,177.370,24.039,153.742
C04269=1089.178,356.732,407.698,177.374,24.047,153.744
C04270=1089.187,357.126,407.642,177.380,24.055,153.745
C04271=1089.196,357.518,407.586,177.385,24.063,153.746
C04272=1089.205,357.911,407.530,177.389,24.071,153.747
C04273=1089.212,358.159,407.495,177.393,24.076,153.748
C04274=1089.217,358.405,407.459,177.396,24.081,153.749
C04275=1089.223,358.653,407.424,177.399,24.086,153.750
C04276=1089.229,358.901,407.388,177.402,24.091,153.750
C04277=1089.236,359.147,407.353,177.406,24.097,153.751
C04278=1089.241,359.396,407.318,177.408,24.102,153.752
C04279=1089.247,359.643,407.282,177.411,24.107,153.753
C04280=1089.253,359.890,407.247,177.414,24.112,153.754
C04281=1089.259,360.138,407.211,177.417,24.117,153.754
C04282=1089.265,360.385,407.177,177.421,24.122,153.755
C04283=1089.271,360.632,407.141,177.423,24.127,153.756
C04284=1089.277,360.880,407.105,177.427,24.133,153.757
C04285=1089.283,361.127,407.070,177.430,24.138,153.758
C04286=1089.289,361.374,407.033,177.433,24.143,153.759
C04287=1089.295,361.622,406.998,177.436,24.148,153.759
C04288=1089.300,361.869,406.962,177.439,24.154,153.760
C04289=1089.306,362.116,406.926,177.442,24.159,153.761
C04290=1089.312,362.364,406.891,177.445,24.164,153.762
C04291=1089.318,362.611,406.855,177.449,24.169,153.763
C04292=1089.324,362.859,406.820,177.451,24.174,153.764
C04293=1089.330,363.106,406.783,177.455,24.180,153.764
C04294=1089.336,363.354,406.747,177.458,24.186,153.765
C04295=1089.342,363.601,406.712,177.460,24.191,153.766
C04296=1089.348,363.848,406.676,177.464,24.196,153.767
C04297=1089.354,364.095,406.640,177.467,24.201,153.768
C04298=1089.359,364.342,406.605,177.471,24.207,153.769
C04299=1089.365,364.590,406.569,177.473,24.212,153.770
C04300=1089.371,364.838,406.533,177.476,24.217,153.770
C04301=1089.378,365.085,406.497,177.480,24.223,153.771
C04302=1089.383,365.332,406.461,177.482,24.228,153.772
C04303=1089.390,365.579,406.425,177.486,24.234,153.773
C04304=1089.396,365.826,406.389,177.489,24.239,153.774
C04305=1089.402,366.074,406.353,177.492,24.245,153.775
C04306=1089.408,366.321,406.317,177.495,24.250,153.776
C04307=1089.413,366.568,406.281,177.498,24.256,153.777
C04308=1089.419,366.815,406.245,177.501,24.261,153.777
C04309=1089.425,367.063,406.209,177.504,24.266,153.778
C04310=1089.431,367.310,406.172,177.507,24.272,153.779
C04311=1089.436,367.557,406.136,177.510,24.278,153.780
C04312=1089.442,367.804,406.100,177.514,24.283,153.781
C04313=1089.448,368.052,406.064,177.516,24.289,153.782
C04314=1089.455,368.299,406.028,177.519,24.295,153.783
C04315=1089.460,368.547,405.991,177.523,24.300,153.784
C04316=1089.466,368.794,405.955,177.526,24.306,153.785
C04317=1089.472,369.041,405.919,177.528,24.311,153.786
C04318=1089.478,369.288,405.883,177.532,24.317,153.787
C04319=1089.484,369.536,405.846,177.535,24.322,153.787
C04320=1089.490,369.783,405.810,177.538,24.328,153.788
C04321=1089.500,370.190,405.750,177.544,24.337,153.790
C04322=1089.510,370.599,405.689,177.549,24.347,153.792
C04323=1089.520,371.007,405.629,177.553,24.356,153.793
C04324=1089.529,371.416,405.569,177.558,24.366,153.795
C04325=1089.535,371.663,405.533,177.561,24.371,153.796
C04326=1089.542,371.910,405.496,177.565,24.377,153.797
C04327=1089.547,372.158,405.459,177.568,24.383,153.798
C04328=1089.554,372.405,405.423,177.571,24.389,153.799
C04329=1089.559,372.652,405.386,177.574,24.394,153.800
C04330=1089.565,372.899,405.349,177.577,24.400,153.801
C04331=1089.572,373.146,405.313,177.580,24.406,153.801
C04332=1089.577,373.393,405.276,177.584,24.412,153.802
C04333=1089.584,373.640,405.240,177.587,24.418,153.804
C04334=1089.590,373.888,405.203,177.590,24.424,153.804
C04335=1089.596,374.135,405.166,177.592,24.429,153.805
C04336=1089.602,374.382,405.130,177.596,24.435,153.807
C04337=1089.608,374.629,405.093,177.599,24.441,153.807
C04338=1089.613,374.877,405.056,177.602,24.447,153.808
C04339=1089.620,375.124,405.019,177.605,24.453,153.810
C04340=1089.625,375.371,404.982,177.608,24.459,153.811
C04341=1089.632,375.618,404.946,177.611,24.465,153.812
C04342=1089.637,375.865,404.908,177.614,24.471,153.813
C04343=1089.643,376.112,404.871,177.617,24.477,153.814
C04344=1089.649,376.359,404.834,177.620,24.483,153.815
C04345=1089.655,376.607,404.797,177.624,24.489,153.816
C04346=1089.661,376.854,404.760,177.627,24.495,153.817
C04347=1089.667,377.100,404.723,177.630,24.501,153.818
C04348=1089.673,377.348,404.686,177.633,24.508,153.819
C04349=1089.679,377.595,404.650,177.636,24.514,153.820
C04350=1089.685,377.842,404.612,177.639,24.519,153.821
C04351=1089.691,378.089,404.575,177.642,24.526,153.822
C04352=1089.697,378.336,404.538,177.645,24.532,153.823
C04353=1089.703,378.583,404.501,177.648,24.538,153.824
C04354=1089.708,378.830,404.464,177.651,24.544,153.825
C04355=1089.714,379.077,404.426,177.655,24.551,153.826
C04356=1089.721,379.325,404.389,177.658,24.557,153.827
C04357=1089.727,379.572,404.352,177.661,24.563,153.829
C04358=1089.733,379.819,404.314,177.664,24.569,153.830
C04359=1089.739,380.066,404.278,177.667,24.576,153.831
C04360=1089.745,380.313,404.240,177.670,24.582,153.832
C04361=1089.751,380.559,404.202,177.674,24.588,153.833
C04362=1089.757,380.807,404.165,177.676,24.594,153.834
C04363=1089.764,381.054,404.128,177.679,24.600,153.835
C04364=1089.769,381.301,404.091,177.682,24.606,153.836
C04365=1089.775,381.548,404.053,177.685,24.613,153.837
C04366=1089.781,381.795,404.015,177.688,24.619,153.838
C04367=1089.788,382.042,403.979,177.692,24.625,153.840
C04368=1089.794,382.289,403.941,177.695,24.632,153.841
C04369=1089.800,382.536,403.903,177.698,24.638,153.842
C04370=1089.806,382.783,403.866,177.701,24.645,153.843
C04371=1089.811,383.030,403.828,177.704,24.651,153.844
C04372=1089.817,383.277,403.790,177.707,24.658,153.845
C04373=1089.823,383.496,403.757,177.711,24.664,153.846
C04374=1089.828,383.713,403.724,177.713,24.669,153.847
C04375=1089.834,383.931,403.690,177.715,24.675,153.848
C04376=1089.838,384.149,403.658,177.719,24.681,153.849
C04377=1089.844,384.367,403.624,177.721,24.687,153.850
C04378=1089.850,384.585,403.590,177.724,24.693,153.852
C04379=1089.854,384.803,403.558,177.727,24.698,153.852
C04380=1089.860,385.021,403.524,177.729,24.704,153.854
C04381=1089.866,385.268,403.486,177.732,24.711,153.855
C04382=1089.872,385.515,403.448,177.736,24.718,153.856
C04383=1089.878,385.762,403.410,177.739,24.724,153.857
C04384=1089.884,386.009,403.372,177.742,24.731,153.858
C04385=1089.890,386.256,403.335,177.745,24.737,153.860
C04386=1089.896,386.503,403.297,177.748,24.744,153.861
C04387=1089.902,386.750,403.259,177.751,24.751,153.862
C04388=1089.908,386.997,403.221,177.754,24.757,153.863
C04389=1089.914,387.244,403.183,177.757,24.764,153.864
C04390=1089.921,387.491,403.145,177.760,24.771,153.866
C04391=1089.926,387.738,403.107,177.763,24.778,153.867
C04392=1089.932,387.985,403.069,177.766,24.784,153.868
C04393=1089.938,388.232,403.031,177.770,24.791,153.869
C04394=1089.945,388.478,402.992,177.773,24.798,153.871
C04395=1089.950,388.725,402.955,177.776,24.804,153.872
C04396=1089.957,388.973,402.917,177.779,24.812,153.873
C04397=1089.963,389.219,402.879,177.783,24.819,153.874
C04398=1089.969,389.465,402.840,177.786,24.825,153.876
C04399=1089.975,389.713,402.802,177.789,24.832,153.877
C04400=1089.981,389.960,402.764,177.792,24.839,153.878
C04401=1089.987,390.207,402.726,177.795,24.846,153.879
C04402=1089.993,390.453,402.687,177.798,24.853,153.881
C04403=1090.000,390.701,402.649,177.801,24.860,153.882
C04404=1090.006,390.947,402.611,177.804,24.867,153.883
C04405=1090.012,391.195,402.572,177.807,24.874,153.885
C04406=1090.018,391.442,402.534,177.811,24.881,153.886
C04407=1090.025,391.688,402.495,177.814,24.888,153.887
C04408=1090.031,391.935,402.458,177.817,24.895,153.889
C04409=1090.037,392.182,402.418,177.820,24.902,153.890
C04410=1090.043,392.429,402.380,177.823,24.909,153.891
C04411=1090.049,392.676,402.342,177.826,24.916,153.893
C04412=1090.055,392.923,402.303,177.828,24.923,153.894
C04413=1090.061,393.170,402.264,177.832,24.931,153.895
C04414=1090.067,393.416,402.227,177.835,24.938,153.897
C04415=1090.073,393.664,402.187,177.838,24.945,153.898
C04416=1090.080,393.910,402.149,177.841,24.952,153.899
C04417=1090.085,394.157,402.110,177.844,24.959,153.901
C04418=1090.091,394.404,402.072,177.848,24.967,153.902
C04419=1090.098,394.651,402.032,177.851,24.974,153.903
C04420=1090.103,394.897,401.994,177.854,24.982,153.905
C04421=1090.110,395.144,401.956,177.857,24.989,153.906
C04422=1090.116,395.391,401.916,177.860,24.996,153.907
C04423=1090.122,395.638,401.878,177.863,25.003,153.909
C04424=1090.128,395.885,401.839,177.867,25.011,153.910
C04425=1090.134,396.132,401.800,177.869,25.018,153.912
C04426=1090.141,396.379,401.761,177.872,25.026,153.913
C04427=1090.147,396.626,401.722,177.875,25.033,153.915
C04428=1090.153,396.872,401.683,177.879,25.041,153.916
C04429=1090.159,397.097,401.647,177.881,25.047,153.917
C04430=1090.164,397.322,401.612,177.884,25.054,153.919
C04431=1090.169,397.546,401.577,177.887,25.061,153.920
C04432=1090.175,397.771,401.541,177.890,25.068,153.921
C04433=1090.181,397.996,401.506,177.893,25.075,153.923
C04434=1090.186,398.221,401.470,177.896,25.082,153.924
C04435=1090.192,398.445,401.434,177.899,25.089,153.925
C04436=1090.198,398.670,401.399,177.902,25.096,153.927
C04437=1090.204,398.917,401.359,177.904,25.103,153.928
C04438=1090.210,399.163,401.321,177.907,25.111,153.930
C04439=1090.216,399.410,401.281,177.911,25.119,153.931
C04440=1090.222,399.657,401.242,177.914,25.126,153.932
C04441=1090.228,399.905,401.202,177.917,25.134,153.934
C04442=1090.234,400.151,401.164,177.920,25.142,153.936
C04443=1090.240,400.398,401.124,177.923,25.150,153.937
C04444=1090.246,400.645,401.085,177.926,25.157,153.938
C04445=1090.253,400.892,401.045,177.929,25.165,153.940
C04446=1090.258,401.138,401.006,177.933,25.173,153.942
C04447=1090.265,401.385,400.967,177.935,25.181,153.943
C04448=1090.271,401.632,400.927,177.938,25.189,153.945
C04449=1090.278,401.878,400.887,177.942,25.197,153.946
C04450=1090.284,402.126,400.848,177.945,25.205,153.948
C04451=1090.289,402.372,400.809,177.949,25.213,153.949
C04452=1090.296,402.619,400.769,177.951,25.221,153.951
C04453=1090.302,402.866,400.729,177.954,25.229,153.952
C04454=1090.308,403.112,400.690,177.958,25.237,153.954
C04455=1090.315,403.359,400.650,177.961,25.245,153.956
C04456=1090.321,403.606,400.611,177.963,25.253,153.957
C04457=1090.327,403.853,400.571,177.967,25.261,153.959
C04458=1090.333,404.100,400.531,177.970,25.269,153.960
C04459=1090.340,404.346,400.491,177.974,25.278,153.962
C04460=1090.345,404.593,400.452,177.976,25.286,153.964
C04461=1090.352,404.839,400.412,177.980,25.294,153.965
C04462=1090.358,405.086,400.372,177.983,25.302,153.967
C04463=1090.364,405.333,400.332,177.986,25.310,153.968
C04464=1090.370,405.580,400.293,177.989,25.319,153.970
C04465=1090.376,405.827,400.253,177.992,25.327,153.972
C04466=1090.383,406.073,400.213,177.996,25.336,153.973
C04467=1090.389,406.320,400.173,177.998,25.344,153.975
C04468=1090.395,406.567,400.133,178.002,25.352,153.977
C04469=1090.402,406.813,400.093,178.005,25.361,153.978
C04470=1090.407,407.061,400.053,178.008,25.370,153.980
C04471=1090.413,407.307,400.013,178.011,25.377,153.982
C04472=1090.420,407.554,399.973,178.015,25.386,153.983
C04473=1090.426,407.800,399.932,178.017,25.395,153.985
C04474=1090.433,408.047,399.892,178.021,25.403,153.987
C04475=1090.439,408.294,399.853,178.024,25.412,153.989
C04476=1090.444,408.541,399.812,178.027,25.421,153.990
C04477=1090.451,408.787,399.772,178.030,25.429,153.992
C04478=1090.457,409.034,399.732,178.033,25.438,153.994
C04479=1090.463,409.281,399.691,178.037,25.447,153.996
C04480=1090.469,409.527,399.651,178.040,25.455,153.997
C04481=1090.475,409.774,399.611,178.043,25.464,153.999
C04482=1090.482,410.020,399.571,178.046,25.473,154.001
C04483=1090.487,410.267,399.530,178.050,25.482,154.003
C04484=1090.494,410.513,399.490,178.052,25.490,154.004
C04485=1090.500,410.739,399.452,178.056,25.499,154.006
C04486=1090.505,410.964,399.415,178.059,25.507,154.008
C04487=1090.511,411.189,399.378,178.061,25.515,154.009
C04488=1090.516,411.414,399.341,178.064,25.523,154.011
C04489=1090.522,411.640,399.305,178.067,25.531,154.013
C04490=1090.528,411.865,399.268,178.070,25.539,154.014
C04491=1090.534,412.090,399.231,178.073,25.547,154.016
C04492=1090.540,412.316,399.194,178.076,25.556,154.018
C04493=1090.546,412.562,399.152,178.079,25.565,154.020
C04494=1090.552,412.808,399.112,178.082,25.574,154.021
C04495=1090.559,413.055,399.072,178.086,25.583,154.023
C04496=1090.564,413.302,399.031,178.089,25.592,154.025
C04497=1090.572,413.548,398.990,178.092,25.601,154.027
C04498=1090.577,413.795,398.949,178.096,25.611,154.029
C04499=1090.584,414.041,398.908,178.098,25.619,154.031
C04500=1090.590,414.288,398.868,178.102,25.629,154.032
C04501=1090.597,414.535,398.827,178.105,25.638,154.034
C04502=1090.603,414.781,398.786,178.109,25.647,154.036
C04503=1090.609,415.028,398.746,178.111,25.656,154.038
C04504=1090.616,415.274,398.704,178.115,25.666,154.040
C04505=1090.622,415.521,398.664,178.118,25.675,154.042
C04506=1090.629,415.767,398.623,178.122,25.685,154.044
C04507=1090.635,416.014,398.581,178.125,25.694,154.046
C04508=1090.641,416.261,398.541,178.128,25.703,154.048
C04509=1090.647,416.507,398.499,178.131,25.713,154.050
C04510=1090.654,416.754,398.458,178.135,25.723,154.052
C04511=1090.660,417.000,398.417,178.138,25.732,154.054
C04512=1090.666,417.246,398.376,178.142,25.742,154.056
C04513=1090.672,417.493,398.334,178.144,25.751,154.058
C04514=1090.679,417.740,398.294,178.147,25.761,154.060
C04515=1090.685,417.986,398.252,178.151,25.771,154.062
C04516=1090.691,418.232,398.211,178.154,25.781,154.064
C04517=1090.698,418.479,398.170,178.158,25.791,154.066
C04518=1090.704,418.725,398.128,178.161,25.800,154.068
C04519=1090.711,418.973,398.087,178.164,25.810,154.070
C04520=1090.717,419.219,398.046,178.167,25.820,154.072
C04521=1090.723,419.465,398.005,178.170,25.830,154.074
C04522=1090.730,419.712,397.963,178.174,25.839,154.076
C04523=1090.736,419.958,397.922,178.177,25.849,154.078
C04524=1090.742,420.205,397.880,178.181,25.859,154.080
C04525=1090.748,420.451,397.838,178.184,25.870,154.082
C04526=1090.755,420.698,397.797,178.187,25.880,154.084
C04527=1090.761,420.944,397.756,178.191,25.890,154.087
C04528=1090.768,421.189,397.713,178.194,25.900,154.089
C04529=1090.774,421.436,397.672,178.197,25.910,154.091
C04530=1090.780,421.682,397.630,178.201,25.920,154.093
C04531=1090.787,421.929,397.589,178.204,25.930,154.095
C04532=1090.794,422.176,397.547,178.207,25.941,154.097
C04533=1090.800,422.422,397.506,178.211,25.951,154.099
C04534=1090.807,422.668,397.463,178.214,25.961,154.101
C04535=1090.813,422.915,397.422,178.217,25.971,154.104
C04536=1090.819,423.162,397.380,178.221,25.982,154.106
C04537=1090.826,423.407,397.338,178.224,25.992,154.108
C04538=1090.832,423.654,397.296,178.227,26.003,154.110
C04539=1090.838,423.900,397.254,178.231,26.013,154.113
C04540=1090.845,424.146,397.212,178.234,26.024,154.115
C04541=1090.850,424.379,397.172,178.237,26.034,154.117
C04542=1090.857,424.612,397.133,178.240,26.043,154.119
C04543=1090.863,424.844,397.093,178.243,26.054,154.121
C04544=1090.869,425.077,397.053,178.247,26.064,154.123
C04545=1090.875,425.310,397.014,178.250,26.074,154.125
C04546=1090.881,425.543,396.973,178.253,26.084,154.128
C04547=1090.887,425.776,396.933,178.256,26.094,154.130
C04548=1090.893,426.008,396.894,178.259,26.104,154.132
C04549=1090.899,426.254,396.851,178.263,26.115,154.134
C04550=1090.906,426.501,396.809,178.266,26.126,154.136
C04551=1090.912,426.747,396.767,178.269,26.137,154.139
C04552=1090.919,426.993,396.725,178.272,26.148,154.141
C04553=1090.926,427.239,396.682,178.276,26.159,154.143
C04554=1090.932,427.485,396.640,178.280,26.170,154.146
C04555=1090.939,427.731,396.597,178.283,26.181,154.148
C04556=1090.945,427.979,396.555,178.286,26.192,154.151
C04557=1090.951,428.225,396.512,178.289,26.203,154.153
C04558=1090.958,428.470,396.470,178.293,26.213,154.155
C04559=1090.965,428.717,396.428,178.297,26.225,154.158
C04560=1090.971,428.963,396.385,178.300,26.236,154.160
C04561=1090.978,429.210,396.342,178.303,26.248,154.163
C04562=1090.984,429.455,396.300,178.306,26.258,154.165
C04563=1090.991,429.701,396.257,178.311,26.270,154.167
C04564=1090.997,429.948,396.214,178.314,26.282,154.170
C04565=1091.004,430.194,396.172,178.317,26.293,154.172
C04566=1091.010,430.440,396.129,178.320,26.304,154.175
C04567=1091.016,430.686,396.086,178.324,26.316,154.177
C04568=1091.023,430.932,396.043,178.327,26.327,154.180
C04569=1091.029,431.179,396.000,178.330,26.339,154.182
C04570=1091.036,431.425,395.957,178.334,26.350,154.185
C04571=1091.043,431.671,395.915,178.338,26.362,154.187
C04572=1091.049,431.917,395.871,178.341,26.374,154.190
C04573=1091.056,432.163,395.829,178.344,26.385,154.192
C04574=1091.062,432.409,395.786,178.348,26.397,154.195
C04575=1091.069,432.655,395.742,178.351,26.409,154.198
C04576=1091.075,432.902,395.699,178.354,26.421,154.200
C04577=1091.082,433.148,395.657,178.358,26.433,154.203
C04578=1091.088,433.394,395.613,178.361,26.445,154.205
C04579=1091.095,433.640,395.570,178.365,26.457,154.208
C04580=1091.102,433.886,395.527,178.368,26.469,154.211
C04581=1091.107,434.132,395.484,178.372,26.481,154.213
C04582=1091.114,434.378,395.441,178.376,26.493,154.216
C04583=1091.121,434.624,395.397,178.379,26.505,154.219
C04584=1091.127,434.870,395.354,178.383,26.518,154.221
C04585=1091.134,435.116,395.310,178.386,26.530,154.224
C04586=1091.140,435.362,395.266,178.389,26.542,154.227
C04587=1091.147,435.609,395.223,178.393,26.554,154.229
C04588=1091.154,435.854,395.180,178.396,26.567,154.232
C04589=1091.160,436.100,395.136,178.400,26.579,154.235
C04590=1091.167,436.346,395.092,178.403,26.591,154.238
C04591=1091.173,436.592,395.050,178.407,26.604,154.240
C04592=1091.180,436.838,395.006,178.410,26.617,154.243
C04593=1091.186,437.084,394.962,178.414,26.629,154.246
C04594=1091.193,437.330,394.918,178.417,26.642,154.249
C04595=1091.200,437.576,394.875,178.421,26.654,154.252
C04596=1091.206,437.822,394.831,178.424,26.667,154.254
C04597=1091.216,438.193,394.765,178.429,26.686,154.259
C04598=1091.227,438.563,394.699,178.435,26.706,154.263
C04599=1091.237,438.933,394.633,178.440,26.725,154.267
C04600=1091.247,439.304,394.567,178.446,26.744,154.272
C04601=1091.253,439.550,394.523,178.449,26.757,154.275
C04602=1091.260,439.796,394.479,178.453,26.770,154.277
C04603=1091.267,440.041,394.435,178.456,26.784,154.280
C04604=1091.274,440.287,394.391,178.459,26.797,154.283
C04605=1091.280,440.533,394.347,178.463,26.810,154.286
C04606=1091.287,440.779,394.303,178.467,26.823,154.289
C04607=1091.294,441.025,394.259,178.470,26.836,154.292
C04608=1091.300,441.271,394.215,178.474,26.850,154.295
C04609=1091.307,441.516,394.170,178.478,26.864,154.298
C04610=1091.314,441.763,394.126,178.481,26.877,154.301
C04611=1091.321,442.008,394.081,178.485,26.891,154.304
C04612=1091.327,442.254,394.038,178.489,26.904,154.307
C04613=1091.334,442.499,393.993,178.492,26.917,154.310
C04614=1091.341,442.746,393.949,178.495,26.931,154.314
C04615=1091.347,442.992,393.904,178.499,26.945,154.317
C04616=1091.354,443.237,393.859,178.503,26.959,154.320
C04617=1091.360,443.483,393.815,178.506,26.973,154.323
C04618=1091.368,443.729,393.770,178.510,26.986,154.326
C04619=1091.374,443.974,393.726,178.514,27.001,154.329
C04620=1091.382,444.220,393.681,178.518,27.015,154.332
C04621=1091.387,444.467,393.636,178.520,27.028,154.336
C04622=1091.394,444.712,393.592,178.524,27.043,154.339
C04623=1091.401,444.958,393.547,178.527,27.057,154.342
C04624=1091.408,445.203,393.502,178.530,27.071,154.345
C04625=1091.415,445.450,393.457,178.533,27.085,154.348
C04626=1091.421,445.695,393.412,178.536,27.098,154.352
C04627=1091.428,445.941,393.368,178.538,27.112,154.355
C04628=1091.435,446.187,393.323,178.540,27.126,154.358
C04629=1091.441,446.432,393.277,178.542,27.140,154.362
C04630=1091.449,446.678,393.233,178.544,27.154,154.365
C04631=1091.456,446.924,393.188,178.545,27.168,154.368
C04632=1091.462,447.170,393.142,178.547,27.182,154.372
C04633=1091.469,447.415,393.098,178.548,27.196,154.375
C04634=1091.476,447.661,393.053,178.550,27.210,154.378
C04635=1091.482,447.907,393.008,178.551,27.223,154.382
C04636=1091.490,448.153,392.962,178.552,27.237,154.385
C04637=1091.496,448.398,392.917,178.553,27.251,154.389
C04638=1091.503,448.644,392.872,178.553,27.265,154.392
C04639=1091.510,448.890,392.827,178.554,27.279,154.396
C04640=1091.516,449.136,392.782,178.554,27.292,154.399
C04641=1091.523,449.381,392.737,178.554,27.306,154.403
C04642=1091.531,449.627,392.692,178.554,27.320,154.406
C04643=1091.538,449.871,392.646,178.554,27.333,154.410
C04644=1091.547,450.118,392.602,178.554,27.346,154.413
C04645=1091.163,450.109,392.419,178.508,27.546,154.468
C04646=1091.153,449.863,392.463,178.508,27.534,154.465
C04647=1091.145,449.618,392.509,178.508,27.520,154.461
C04648=1091.139,449.372,392.554,178.508,27.506,154.458
C04649=1091.132,449.128,392.599,178.507,27.492,154.455
C04650=1091.125,448.881,392.644,178.507,27.479,154.451
C04651=1091.119,448.636,392.689,178.506,27.464,154.448
C04652=1091.111,448.390,392.735,178.505,27.451,154.444
C04653=1091.105,448.144,392.780,178.505,27.437,154.441
C04654=1091.098,447.899,392.825,178.504,27.423,154.437
C04655=1091.092,447.652,392.870,178.503,27.409,154.434
C04656=1091.085,447.408,392.916,178.501,27.395,154.430
C04657=1091.077,447.162,392.961,178.500,27.381,154.427
C04658=1091.071,446.915,393.006,178.498,27.367,154.424
C04659=1091.064,446.670,393.051,178.497,27.354,154.420
C04660=1091.057,446.424,393.096,178.495,27.340,154.417
C04661=1091.051,446.178,393.141,178.492,27.325,154.414
C04662=1091.043,445.932,393.186,178.490,27.312,154.410
C04663=1091.037,445.686,393.231,178.488,27.297,154.407
C04664=1091.031,445.441,393.275,178.485,27.284,154.404
C04665=1091.023,445.196,393.321,178.482,27.269,154.400
C04666=1091.016,444.950,393.365,178.479,27.255,154.397
C04667=1091.009,444.704,393.410,178.476,27.241,154.394
C04668=1091.003,444.458,393.455,178.472,27.227,154.391
C04669=1090.996,444.212,393.500,178.468,27.213,154.388
C04670=1090.989,443.966,393.545,178.465,27.199,154.384
C04671=1090.982,443.721,393.589,178.461,27.185,154.381
C04672=1090.975,443.475,393.634,178.457,27.171,154.378
C04673=1090.969,443.229,393.678,178.453,27.157,154.375
C04674=1090.963,442.983,393.723,178.450,27.144,154.372
C04675=1090.955,442.737,393.768,178.446,27.130,154.369
C04676=1090.949,442.492,393.813,178.443,27.116,154.366
C04677=1090.942,442.246,393.856,178.439,27.102,154.363
C04678=1090.935,442.000,393.901,178.436,27.089,154.359
C04679=1090.928,441.754,393.945,178.432,27.075,154.356
C04680=1090.922,441.509,393.990,178.428,27.062,154.353
C04681=1090.915,441.263,394.034,178.425,27.048,154.350
C04682=1090.908,441.017,394.079,178.421,27.035,154.347
C04683=1090.901,440.771,394.122,178.417,27.021,154.344
C04684=1090.895,440.525,394.167,178.414,27.008,154.341
C04685=1090.888,440.279,394.211,178.410,26.995,154.338
C04686=1090.881,440.033,394.256,178.406,26.982,154.335
C04687=1090.875,439.787,394.300,178.402,26.968,154.332
C04688=1090.868,439.541,394.343,178.398,26.955,154.330
C04689=1090.862,439.295,394.387,178.395,26.942,154.327
C04690=1090.851,438.937,394.452,178.390,26.923,154.322
C04691=1090.841,438.579,394.515,178.385,26.904,154.318
C04692=1090.832,438.221,394.579,178.379,26.886,154.314
C04693=1090.821,437.862,394.643,178.375,26.867,154.310
C04694=1090.815,437.616,394.687,178.371,26.854,154.307
C04695=1090.809,437.370,394.731,178.367,26.842,154.304
C04696=1090.801,437.125,394.774,178.363,26.829,154.301
C04697=1090.795,436.879,394.818,178.360,26.816,154.299
C04698=1090.789,436.633,394.862,178.356,26.804,154.296
C04699=1090.782,436.387,394.906,178.353,26.791,154.293
C04700=1090.775,436.141,394.949,178.349,26.779,154.290
C04701=1090.769,435.895,394.993,178.346,26.766,154.288
C04702=1090.762,435.649,395.037,178.342,26.754,154.285
C04703=1090.755,435.403,395.080,178.339,26.742,154.282
C04704=1090.749,435.157,395.123,178.334,26.729,154.279
C04705=1090.742,434.911,395.167,178.331,26.717,154.277
C04706=1090.735,434.665,395.210,178.327,26.704,154.274
C04707=1090.729,434.419,395.253,178.324,26.692,154.271
C04708=1090.723,434.173,395.297,178.321,26.680,154.269
C04709=1090.716,433.927,395.340,178.317,26.668,154.266
C04710=1090.709,433.680,395.383,178.314,26.656,154.263
C04711=1090.703,433.434,395.427,178.310,26.644,154.261
C04712=1090.696,433.188,395.470,178.306,26.631,154.258
C04713=1090.690,432.942,395.514,178.303,26.620,154.255
C04714=1090.683,432.696,395.556,178.300,26.608,154.253
C04715=1090.677,432.450,395.600,178.296,26.596,154.250
C04716=1090.670,432.204,395.642,178.293,26.584,154.248
C04717=1090.664,431.958,395.686,178.289,26.573,154.245
C04718=1090.657,431.712,395.729,178.285,26.561,154.243
C04719=1090.651,431.465,395.772,178.282,26.549,154.240
C04720=1090.644,431.220,395.815,178.279,26.537,154.237
C04721=1090.637,430.973,395.858,178.275,26.526,154.235
C04722=1090.631,430.727,395.901,178.271,26.514,154.232
C04723=1090.624,430.481,395.943,178.268,26.503,154.230
C04724=1090.618,430.235,395.986,178.265,26.491,154.227
C04725=1090.611,429.989,396.029,178.261,26.479,154.225
C04726=1090.604,429.743,396.072,178.258,26.468,154.222
C04727=1090.598,429.496,396.115,178.254,26.457,154.220
C04728=1090.592,429.251,396.157,178.251,26.445,154.218
C04729=1090.585,429.004,396.200,178.247,26.434,154.215
C04730=1090.579,428.758,396.243,178.244,26.423,154.213
C04731=1090.572,428.511,396.285,178.240,26.412,154.210
C04732=1090.565,428.265,396.328,178.237,26.401,154.208
C04733=1090.559,428.019,396.370,178.234,26.390,154.206
C04734=1090.553,427.773,396.413,178.229,26.378,154.203
C04735=1090.546,427.527,396.456,178.226,26.367,154.201
C04736=1090.539,427.280,396.497,178.223,26.356,154.198
C04737=1090.533,427.034,396.540,178.220,26.345,154.196
C04738=1090.526,426.788,396.582,178.216,26.334,154.194
C04739=1090.520,426.542,396.625,178.213,26.324,154.191
C04740=1090.513,426.296,396.667,178.210,26.313,154.189
C04741=1090.507,426.049,396.709,178.206,26.302,154.187
C04742=1090.501,425.816,396.749,178.203,26.291,154.184
C04743=1090.494,425.583,396.789,178.199,26.281,154.182
C04744=1090.488,425.350,396.829,178.196,26.271,154.180
C04745=1090.483,425.117,396.869,178.192,26.261,154.178
C04746=1090.476,424.883,396.909,178.190,26.251,154.176
C04747=1090.470,424.650,396.949,178.186,26.241,154.174
C04748=1090.465,424.416,396.989,178.183,26.231,154.172
C04749=1090.459,424.183,397.029,178.180,26.221,154.169
C04750=1090.452,423.937,397.071,178.176,26.210,154.167
C04751=1090.445,423.690,397.113,178.173,26.199,154.165
C04752=1090.439,423.445,397.155,178.169,26.189,154.163
C04753=1090.433,423.198,397.197,178.166,26.178,154.161
C04754=1090.427,422.951,397.239,178.163,26.168,154.158
C04755=1090.420,422.705,397.281,178.159,26.157,154.156
C04756=1090.414,422.459,397.323,178.156,26.147,154.154
C04757=1090.407,422.212,397.364,178.153,26.137,154.152
C04758=1090.401,421.966,397.407,178.149,26.127,154.150
C04759=1090.394,421.720,397.448,178.146,26.116,154.147
C04760=1090.388,421.474,397.489,178.143,26.106,154.145
C04761=1090.381,421.227,397.531,178.140,26.096,154.143
C04762=1090.375,420.981,397.573,178.136,26.086,154.141
C04763=1090.368,420.734,397.615,178.133,26.076,154.139
C04764=1090.362,420.488,397.656,178.130,26.066,154.137
C04765=1090.355,420.242,397.698,178.126,26.056,154.135
C04766=1090.349,419.995,397.739,178.123,26.046,154.133
C04767=1090.343,419.748,397.781,178.119,26.036,154.131
C04768=1090.337,419.502,397.823,178.116,26.026,154.129
C04769=1090.329,419.256,397.864,178.112,26.016,154.126
C04770=1090.323,419.009,397.905,178.109,26.006,154.124
C04771=1090.317,418.762,397.947,178.106,25.996,154.122
C04772=1090.311,418.516,397.988,178.103,25.986,154.120
C04773=1090.304,418.270,398.029,178.099,25.976,154.118
C04774=1090.298,418.023,398.070,178.096,25.967,154.116
C04775=1090.292,417.777,398.112,178.092,25.957,154.114
C04776=1090.286,417.530,398.153,178.089,25.947,154.112
C04777=1090.279,417.284,398.195,178.086,25.938,154.110
C04778=1090.273,417.038,398.236,178.083,25.928,154.108
C04779=1090.267,416.791,398.277,178.079,25.918,154.106
C04780=1090.260,416.544,398.318,178.076,25.908,154.104
C04781=1090.254,416.298,398.359,178.072,25.899,154.102
C04782=1090.248,416.051,398.400,178.070,25.889,154.100
C04783=1090.241,415.805,398.441,178.066,25.880,154.098
C04784=1090.235,415.558,398.483,178.063,25.871,154.096
C04785=1090.228,415.311,398.523,178.059,25.861,154.094
C04786=1090.222,415.065,398.565,178.056,25.852,154.093
C04787=1090.216,414.818,398.605,178.053,25.843,154.091
C04788=1090.209,414.572,398.646,178.049,25.833,154.089
C04789=1090.203,414.325,398.687,178.046,25.824,154.087
C04790=1090.196,414.079,398.728,178.043,25.815,154.085
C04791=1090.191,413.832,398.769,178.040,25.806,154.083
C04792=1090.183,413.586,398.810,178.036,25.796,154.081
C04793=1090.178,413.339,398.851,178.033,25.787,154.079
C04794=1090.171,413.092,398.891,178.030,25.778,154.077
C04795=1090.165,412.847,398.932,178.026,25.769,154.076
C04796=1090.158,412.599,398.973,178.023,25.760,154.074
C04797=1090.152,412.352,399.013,178.020,25.751,154.072
C04798=1090.146,412.127,399.050,178.017,25.742,154.070
C04799=1090.140,411.902,399.087,178.014,25.734,154.068
C04800=1090.135,411.676,399.125,178.011,25.726,154.067
C04801=1090.129,411.449,399.162,178.008,25.717,154.065
C04802=1090.124,411.224,399.199,178.005,25.709,154.063
C04803=1090.118,410.999,399.236,178.002,25.701,154.062
C04804=1090.112,410.772,399.273,177.999,25.693,154.060
C04805=1090.106,410.547,399.310,177.996,25.685,154.059
C04806=1090.100,410.301,399.350,177.993,25.676,154.057
C04807=1090.094,410.053,399.391,177.989,25.667,154.055
C04808=1090.087,409.807,399.431,177.986,25.658,154.053
C04809=1090.081,409.560,399.472,177.983,25.650,154.051
C04810=1090.075,409.314,399.512,177.980,25.641,154.050
C04811=1090.069,409.067,399.552,177.977,25.632,154.048
C04812=1090.063,408.821,399.593,177.974,25.624,154.046
C04813=1090.056,408.574,399.633,177.970,25.614,154.044
C04814=1090.051,408.327,399.674,177.967,25.606,154.043
C04815=1090.044,408.081,399.714,177.964,25.597,154.041
C04816=1090.038,407.834,399.754,177.961,25.589,154.039
C04817=1090.031,407.588,399.794,177.957,25.580,154.037
C04818=1090.026,407.340,399.834,177.955,25.572,154.036
C04819=1090.020,407.094,399.874,177.951,25.563,154.034
C04820=1090.013,406.847,399.914,177.948,25.555,154.032
C04821=1090.007,406.601,399.954,177.945,25.546,154.031
C04822=1090.001,406.354,399.995,177.942,25.538,154.029
C04823=1089.995,406.107,400.034,177.938,25.529,154.027
C04824=1089.988,405.860,400.074,177.935,25.521,154.026
C04825=1089.982,405.614,400.114,177.932,25.512,154.024
C04826=1089.976,405.367,400.154,177.929,25.504,154.022
C04827=1089.969,405.120,400.194,177.925,25.496,154.021
C04828=1089.963,404.874,400.234,177.922,25.487,154.019
C04829=1089.957,404.627,400.273,177.920,25.479,154.017
C04830=1089.950,404.380,400.314,177.916,25.471,154.016
C04831=1089.944,404.133,400.353,177.913,25.463,154.014
C04832=1089.938,403.886,400.393,177.909,25.454,154.012
C04833=1089.932,403.639,400.433,177.906,25.446,154.011
C04834=1089.926,403.394,400.472,177.904,25.438,154.009
C04835=1089.920,403.146,400.512,177.900,25.430,154.008
C04836=1089.914,402.900,400.552,177.897,25.422,154.006
C04837=1089.908,402.653,400.591,177.893,25.414,154.005
C04838=1089.902,402.406,400.631,177.890,25.406,154.003
C04839=1089.895,402.159,400.671,177.888,25.398,154.001
C04840=1089.888,401.912,400.710,177.884,25.390,154.000
C04841=1089.882,401.665,400.749,177.881,25.382,153.998
C04842=1089.877,401.419,400.789,177.878,25.374,153.997
C04843=1089.870,401.172,400.828,177.874,25.366,153.995
C04844=1089.864,400.925,400.868,177.872,25.358,153.994
C04845=1089.858,400.678,400.907,177.869,25.351,153.992
C04846=1089.851,400.432,400.947,177.865,25.342,153.991
C04847=1089.846,400.185,400.986,177.862,25.335,153.989
C04848=1089.840,399.938,401.025,177.859,25.327,153.987
C04849=1089.834,399.691,401.065,177.856,25.319,153.986
C04850=1089.827,399.444,401.104,177.852,25.311,153.985
C04851=1089.821,399.198,401.143,177.849,25.304,153.983
C04852=1089.815,398.951,401.182,177.847,25.296,153.981
C04853=1089.809,398.703,401.222,177.843,25.288,153.980
C04854=1089.803,398.478,401.257,177.841,25.281,153.979
C04855=1089.798,398.254,401.293,177.838,25.274,153.977
C04856=1089.792,398.028,401.328,177.835,25.267,153.976
C04857=1089.786,397.803,401.364,177.832,25.260,153.975
C04858=1089.780,397.578,401.400,177.829,25.253,153.973
C04859=1089.776,397.353,401.436,177.826,25.247,153.972
C04860=1089.770,397.128,401.471,177.823,25.240,153.971
C04861=1089.764,396.902,401.507,177.820,25.233,153.969
C04862=1089.757,396.656,401.546,177.817,25.225,153.968
C04863=1089.751,396.409,401.585,177.814,25.217,153.966
C04864=1089.745,396.162,401.624,177.811,25.210,153.965
C04865=1089.739,395.916,401.663,177.807,25.202,153.964
C04866=1089.733,395.668,401.702,177.805,25.195,153.962
C04867=1089.727,395.422,401.740,177.802,25.188,153.961
C04868=1089.721,395.175,401.780,177.799,25.180,153.959
C04869=1089.714,394.928,401.818,177.796,25.173,153.958
C04870=1089.709,394.681,401.857,177.792,25.165,153.957
C04871=1089.702,394.434,401.896,177.789,25.158,153.955
C04872=1089.697,394.188,401.935,177.786,25.151,153.954
C04873=1089.690,393.940,401.973,177.783,25.144,153.952
C04874=1089.684,393.693,402.012,177.780,25.136,153.951
C04875=1089.678,393.447,402.051,177.777,25.129,153.950
C04876=1089.671,393.199,402.089,177.773,25.122,153.948
C04877=1089.666,392.953,402.128,177.770,25.115,153.947
C04878=1089.659,392.706,402.167,177.767,25.108,153.946
C04879=1089.654,392.459,402.205,177.764,25.100,153.944
C04880=1089.647,392.212,402.244,177.761,25.093,153.943
C04881=1089.641,391.966,402.282,177.758,25.086,153.942
C04882=1089.635,391.718,402.321,177.755,25.079,153.940
C04883=1089.629,391.472,402.359,177.751,25.072,153.939
C04884=1089.623,391.225,402.398,177.748,25.065,153.938
C04885=1089.617,390.978,402.435,177.745,25.058,153.936
C04886=1089.610,390.731,402.474,177.742,25.051,153.935
C04887=1089.605,390.484,402.513,177.739,25.044,153.934
C04888=1089.598,390.237,402.551,177.736,25.037,153.932
C04889=1089.592,389.991,402.589,177.733,25.030,153.931
C04890=1089.585,389.743,402.627,177.730,25.023,153.930
C04891=1089.580,389.496,402.665,177.727,25.016,153.929
C04892=1089.573,389.250,402.704,177.723,25.009,153.927
C04893=1089.567,389.003,402.742,177.719,25.002,153.926
C04894=1089.562,388.756,402.780,177.717,24.995,153.925
C04895=1089.555,388.508,402.818,177.713,24.988,153.924
C04896=1089.549,388.262,402.857,177.710,24.982,153.922
C04897=1089.543,388.016,402.894,177.707,24.975,153.921
C04898=1089.537,387.768,402.932,177.704,24.968,153.920
C04899=1089.531,387.521,402.970,177.701,24.961,153.919
C04900=1089.525,387.275,403.008,177.698,24.955,153.917
C04901=1089.518,387.027,403.046,177.695,24.948,153.916
C04902=1089.512,386.780,403.084,177.692,24.941,153.915
C04903=1089.507,386.534,403.123,177.689,24.934,153.914
C04904=1089.500,386.287,403.161,177.686,24.928,153.912
C04905=1089.494,386.040,403.199,177.682,24.921,153.911
C04906=1089.488,385.793,403.237,177.679,24.914,153.910
C04907=1089.482,385.546,403.275,177.676,24.908,153.909
C04908=1089.476,385.299,403.312,177.673,24.901,153.908
C04909=1089.470,385.052,403.350,177.670,24.894,153.906
C04910=1089.465,384.833,403.383,177.667,24.888,153.905
C04911=1089.460,384.614,403.417,177.664,24.882,153.904
C04912=1089.454,384.396,403.450,177.661,24.877,153.903
C04913=1089.449,384.177,403.484,177.659,24.871,153.902
C04914=1089.444,383.959,403.517,177.656,24.865,153.901
C04915=1089.439,383.740,403.551,177.653,24.859,153.900
C04916=1089.433,383.522,403.584,177.651,24.853,153.899
C04917=1089.428,383.304,403.617,177.647,24.847,153.898
C04918=1089.421,383.057,403.655,177.644,24.841,153.897
C04919=1089.415,382.810,403.693,177.641,24.834,153.896
C04920=1089.410,382.563,403.730,177.638,24.828,153.894
C04921=1089.404,382.316,403.767,177.635,24.821,153.893
C04922=1089.397,382.069,403.805,177.632,24.815,153.892
C04923=1089.392,381.821,403.842,177.629,24.809,153.891
C04924=1089.386,381.575,403.880,177.625,24.802,153.890
C04925=1089.379,381.328,403.917,177.623,24.796,153.889
C04926=1089.374,381.081,403.954,177.620,24.790,153.888
C04927=1089.367,380.833,403.993,177.617,24.784,153.887
C04928=1089.361,380.587,404.030,177.613,24.777,153.886
C04929=1089.355,380.340,404.067,177.610,24.771,153.884
C04930=1089.349,380.093,404.105,177.607,24.765,153.883
C04931=1089.343,379.845,404.142,177.604,24.758,153.882
C04932=1089.337,379.599,404.179,177.601,24.752,153.881
C04933=1089.331,379.351,404.216,177.598,24.746,153.880
C04934=1089.325,379.104,404.254,177.594,24.740,153.879
C04935=1089.319,378.857,404.291,177.591,24.733,153.878
C04936=1089.312,378.610,404.328,177.588,24.727,153.877
C04937=1089.307,378.363,404.365,177.586,24.721,153.876
C04938=1089.301,378.116,404.402,177.582,24.715,153.875
C04939=1089.295,377.869,404.439,177.579,24.709,153.874
C04940=1089.289,377.622,404.476,177.576,24.703,153.872
C04941=1089.283,377.375,404.514,177.573,24.696,153.871
C04942=1089.277,377.128,404.551,177.570,24.690,153.870
C04943=1089.271,376.881,404.588,177.566,24.684,153.869
C04944=1089.266,376.633,404.625,177.563,24.678,153.868
C04945=1089.259,376.387,404.662,177.560,24.672,153.867
C04946=1089.253,376.139,404.699,177.557,24.666,153.866
C04947=1089.247,375.891,404.736,177.554,24.660,153.865
C04948=1089.241,375.644,404.773,177.551,24.654,153.864
C04949=1089.235,375.398,404.810,177.548,24.648,153.863
C04950=1089.229,375.151,404.847,177.545,24.642,153.862
C04951=1089.224,374.904,404.884,177.541,24.635,153.861
C04952=1089.218,374.657,404.921,177.539,24.630,153.860
C04953=1089.212,374.410,404.957,177.536,24.624,153.859
C04954=1089.206,374.162,404.994,177.532,24.618,153.858
C04955=1089.200,373.915,405.031,177.529,24.612,153.857
C04956=1089.194,373.668,405.068,177.526,24.606,153.856
C04957=1089.188,373.421,405.104,177.523,24.600,153.855
C04958=1089.181,373.174,405.140,177.520,24.594,153.854
C04959=1089.176,372.926,405.178,177.517,24.589,153.853
C04960=1089.169,372.679,405.214,177.514,24.583,153.852
C04961=1089.163,372.432,405.250,177.510,24.577,153.851
C04962=1089.158,372.185,405.287,177.507,24.571,153.850
C04963=1089.151,371.938,405.324,177.505,24.565,153.849
C04964=1089.146,371.690,405.361,177.501,24.560,153.848
C04965=1089.139,371.443,405.397,177.498,24.554,153.847
C04966=1089.129,371.033,405.458,177.493,24.544,153.845
C04967=1089.120,370.625,405.519,177.488,24.535,153.844
C04968=1089.109,370.216,405.578,177.482,24.525,153.842
C04969=1089.100,369.807,405.639,177.477,24.515,153.841
C04970=1089.094,369.559,405.674,177.475,24.511,153.840
C04971=1089.088,369.312,405.712,177.471,24.505,153.839
C04972=1089.082,369.065,405.748,177.468,24.499,153.838
C04973=1089.076,368.817,405.784,177.465,24.493,153.837
C04974=1089.069,368.570,405.820,177.462,24.488,153.836
C04975=1089.064,368.323,405.857,177.459,24.482,153.835
C04976=1089.058,368.076,405.893,177.456,24.476,153.834
C04977=1089.052,367.829,405.929,177.452,24.470,153.833
C04978=1089.046,367.581,405.966,177.450,24.465,153.832
C04979=1089.040,367.334,406.002,177.447,24.460,153.831
C04980=1089.034,367.087,406.038,177.443,24.454,153.830
C04981=1089.029,366.840,406.074,177.440,24.448,153.829
C04982=1089.022,366.593,406.110,177.437,24.443,153.829
C04983=1089.017,366.345,406.146,177.434,24.437,153.828
C04984=1089.011,366.097,406.183,177.431,24.431,153.827
C04985=1089.005,365.851,406.218,177.428,24.427,153.826
C04986=1088.999,365.603,406.255,177.425,24.421,153.825
C04987=1088.993,365.356,406.290,177.421,24.415,153.824
C04988=1088.987,365.108,406.326,177.418,24.410,153.823
C04989=1088.980,364.861,406.362,177.416,24.405,153.822
C04990=1088.976,364.614,406.398,177.412,24.399,153.821
C04991=1088.970,364.366,406.434,177.409,24.393,153.820
C04992=1088.963,364.119,406.471,177.406,24.389,153.820
C04993=1088.957,363.871,406.506,177.403,24.383,153.819
C04994=1088.952,363.624,406.542,177.400,24.377,153.818
C04995=1088.946,363.377,406.578,177.397,24.372,153.817
C04996=1088.940,363.130,406.614,177.394,24.367,153.816
C04997=1088.933,362.882,406.650,177.390,24.361,153.815
C04998=1088.928,362.635,406.685,177.388,24.356,153.814
C04999=1088.921,362.388,406.720,177.384,24.351,153.814
C05000=1088.915,362.141,406.757,177.381,24.345,153.813
C05001=1088.910,361.894,406.792,177.379,24.340,153.812
C05002=1088.904,361.646,406.828,177.375,24.335,153.811
C05003=1088.897,361.398,406.863,177.372,24.330,153.810
C05004=1088.892,361.151,406.899,177.369,24.325,153.809
C05005=1088.886,360.904,406.934,177.366,24.319,153.809
C05006=1088.880,360.656,406.970,177.362,24.314,153.808
C05007=1088.875,360.409,407.006,177.360,24.309,153.807
C05008=1088.869,360.161,407.041,177.356,24.304,153.806
C05009=1088.862,359.914,407.077,177.353,24.298,153.805
C05010=1088.857,359.667,407.112,177.350,24.293,153.804
C05011=1088.850,359.419,407.148,177.347,24.288,153.804
C05012=1088.844,359.172,407.183,177.344,24.283,153.803
C05013=1088.839,358.925,407.219,177.341,24.278,153.802
C05014=1088.833,358.677,407.254,177.338,24.272,153.801
C05015=1088.826,358.430,407.289,177.335,24.268,153.801
C05016=1088.821,358.183,407.325,177.331,24.262,153.800
C05017=1088.815,357.935,407.361,177.328,24.257,153.799
C05018=1088.806,357.541,407.417,177.323,24.249,153.798
C05019=1088.795,357.148,407.473,177.319,24.241,153.796
C05020=1088.786,356.754,407.529,177.313,24.233,153.795
C05021=1088.777,356.361,407.585,177.309,24.225,153.794
C05022=1088.772,356.112,407.620,177.306,24.220,153.793
C05023=1088.765,355.865,407.655,177.303,24.215,153.792
C05024=1088.760,355.618,407.690,177.299,24.209,153.792
C05025=1088.753,355.370,407.726,177.296,24.205,153.791
C05026=1088.748,355.123,407.760,177.293,24.200,153.790
C05027=1088.742,354.875,407.796,177.290,24.195,153.789
C05028=1088.736,354.628,407.831,177.287,24.190,153.788
C05029=1088.730,354.380,407.866,177.284,24.185,153.788
C05030=1088.724,354.133,407.901,177.281,24.180,153.787
C05031=1088.719,353.885,407.936,177.277,24.175,153.786
C05032=1088.712,353.638,407.971,177.275,24.170,153.785
C05033=1088.707,353.390,408.006,177.271,24.165,153.785
C05034=1088.700,353.144,408.041,177.269,24.160,153.784
C05035=1088.695,352.896,408.075,177.265,24.155,153.783
C05036=1088.689,352.648,408.111,177.263,24.150,153.782
C05037=1088.683,352.401,408.145,177.259,24.145,153.782
C05038=1088.677,352.153,408.181,177.256,24.141,153.781
C05039=1088.672,351.906,408.215,177.253,24.136,153.780
C05040=1088.665,351.659,408.250,177.250,24.131,153.780
C05041=1088.660,351.411,408.285,177.247,24.126,153.779
C05042=1088.653,351.163,408.319,177.243,24.121,153.778
C05043=1088.648,350.916,408.354,177.241,24.117,153.777
C05044=1088.641,350.668,408.389,177.237,24.112,153.777
C05045=1088.636,350.421,408.423,177.235,24.107,153.776
C05046=1088.630,350.174,408.458,177.231,24.102,153.775
C05047=1088.624,349.926,408.493,177.228,24.097,153.775
C05048=1088.618,349.678,408.527,177.225,24.092,153.774
C05049=1088.612,349.430,408.562,177.222,24.088,153.773
C05050=1088.607,349.183,408.597,177.219,24.083,153.773
C05051=1088.601,348.936,408.631,177.216,24.078,153.772
C05052=1088.595,348.688,408.666,177.212,24.074,153.771
C05053=1088.589,348.440,408.700,177.210,24.069,153.770
C05054=1088.583,348.193,408.734,177.206,24.064,153.770
C05055=1088.577,347.946,408.770,177.204,24.060,153.769
C05056=1088.571,347.698,408.804,177.200,24.055,153.768
C05057=1088.565,347.450,408.838,177.197,24.050,153.768
C05058=1088.560,347.203,408.873,177.194,24.045,153.767
C05059=1088.554,346.955,408.907,177.191,24.041,153.766
C05060=1088.548,346.708,408.941,177.189,24.036,153.766
C05061=1088.542,346.460,408.976,177.185,24.031,153.765
C05062=1088.536,346.212,409.010,177.182,24.027,153.764
C05063=1088.531,345.965,409.044,177.179,24.022,153.764
C05064=1088.525,345.717,409.079,177.176,24.017,153.763
C05065=1088.519,345.470,409.113,177.173,24.013,153.762
C05066=1088.513,345.222,409.147,177.170,24.008,153.762
C05067=1088.507,344.975,409.181,177.166,24.003,153.761
C05068=1088.502,344.727,409.216,177.164,23.999,153.760
C05069=1088.496,344.479,409.251,177.160,23.994,153.760
C05070=1088.486,344.088,409.304,177.155,23.987,153.759
C05071=1088.477,343.698,409.358,177.150,23.980,153.758
C05072=1088.468,343.306,409.412,177.145,23.973,153.757
C05073=1088.458,342.915,409.466,177.141,23.966,153.756
C05074=1088.452,342.668,409.500,177.138,23.961,153.755
C05075=1088.446,342.421,409.534,177.135,23.957,153.754
C05076=1088.441,342.173,409.567,177.132,23.952,153.754
C05077=1088.436,341.925,409.602,177.129,23.948,153.753
C05078=1088.429,341.677,409.636,177.125,23.943,153.752
C05079=1088.423,341.430,409.670,177.123,23.939,153.752
C05080=1088.418,341.182,409.704,177.120,23.935,153.751
C05081=1088.412,340.935,409.738,177.116,23.930,153.751
C05082=1088.406,340.687,409.772,177.114,23.926,153.750
C05083=1088.400,340.439,409.805,177.110,23.921,153.749
C05084=1088.394,340.191,409.839,177.107,23.917,153.749
C05085=1088.388,339.944,409.873,177.105,23.913,153.748
C05086=1088.382,339.696,409.907,177.101,23.908,153.747
C05087=1088.377,339.449,409.941,177.098,23.904,153.747
C05088=1088.371,339.201,409.974,177.095,23.899,153.746
C05089=1088.365,338.954,410.008,177.092,23.895,153.746
C05090=1088.359,338.705,410.042,177.089,23.891,153.745
C05091=1088.353,338.458,410.076,177.086,23.886,153.744
C05092=1088.348,338.210,410.109,177.083,23.882,153.744
C05093=1088.342,337.963,410.143,177.080,23.877,153.743
C05094=1088.336,337.715,410.177,177.077,23.873,153.743
C05095=1088.330,337.467,410.210,177.074,23.868,153.742
C05096=1088.324,337.220,410.244,177.070,23.864,153.741
C05097=1088.319,336.972,410.277,177.067,23.860,153.741
C05098=1088.312,336.724,410.311,177.065,23.856,153.740
C05099=1088.306,336.476,410.345,177.061,23.851,153.740
C05100=1088.301,336.228,410.378,177.058,23.847,153.739
C05101=1088.294,335.981,410.412,177.055,23.843,153.738
C05102=1088.289,335.733,410.445,177.052,23.838,153.738
C05103=1088.283,335.485,410.478,177.049,23.834,153.737
C05104=1088.277,335.238,410.512,177.046,23.830,153.737
C05105=1088.272,334.990,410.546,177.043,23.826,153.736
C05106=1088.266,334.743,410.578,177.040,23.822,153.736
C05107=1088.260,334.495,410.612,177.037,23.817,153.735
C05108=1088.254,334.247,410.645,177.034,23.813,153.734
C05109=1088.249,334.000,410.679,177.031,23.809,153.734
C05110=1088.243,333.752,410.712,177.028,23.804,153.733
C05111=1088.237,333.504,410.745,177.024,23.800,153.733
C05112=1088.231,333.256,410.778,177.022,23.796,153.732
C05113=1088.226,333.008,410.812,177.019,23.792,153.732
C05114=1088.219,332.761,410.845,177.016,23.788,153.731
C05115=1088.213,332.513,410.879,177.012,23.783,153.731
C05116=1088.208,332.265,410.912,177.010,23.779,153.730
C05117=1088.202,332.018,410.945,177.007,23.775,153.729
C05118=1088.196,331.770,410.978,177.003,23.771,153.729
C05119=1088.190,331.522,411.011,177.000,23.767,153.728
C05120=1088.184,331.274,411.044,176.997,23.763,153.728
C05121=1088.179,331.027,411.077,176.994,23.758,153.727
C05122=1088.168,330.630,411.130,176.990,23.752,153.726
C05123=1088.159,330.233,411.183,176.985,23.746,153.726
C05124=1088.150,329.836,411.236,176.980,23.739,153.725
C05125=1088.140,329.440,411.288,176.975,23.733,153.724
C05126=1088.134,329.192,411.322,176.972,23.729,153.723
C05127=1088.128,328.944,411.354,176.969,23.725,153.723
C05128=1088.123,328.696,411.387,176.965,23.721,153.723
C05129=1088.117,328.448,411.420,176.962,23.717,153.722
C05130=1088.110,328.200,411.453,176.960,23.712,153.721
C05131=1088.105,327.953,411.486,176.957,23.709,153.721
C05132=1088.098,327.705,411.519,176.953,23.704,153.720
C05133=1088.093,327.456,411.551,176.950,23.701,153.720
C05134=1088.088,327.210,411.584,176.947,23.697,153.719
C05135=1088.081,326.962,411.616,176.945,23.693,153.719
C05136=1088.076,326.714,411.650,176.941,23.689,153.718
C05137=1088.070,326.466,411.682,176.938,23.684,153.718
C05138=1088.064,326.218,411.715,176.935,23.681,153.717
C05139=1088.058,325.970,411.748,176.932,23.677,153.717
C05140=1088.052,325.722,411.780,176.929,23.672,153.716
C05141=1088.047,325.475,411.813,176.926,23.669,153.716
C05142=1088.041,325.227,411.846,176.923,23.665,153.715
C05143=1088.035,324.979,411.878,176.920,23.661,153.715
C05144=1088.029,324.731,411.911,176.917,23.657,153.714
C05145=1088.023,324.483,411.943,176.914,23.653,153.714
C05146=1088.017,324.235,411.976,176.911,23.649,153.713
C05147=1088.012,323.988,412.008,176.908,23.645,153.713
C05148=1088.006,323.740,412.041,176.905,23.641,153.712
C05149=1088.000,323.492,412.073,176.901,23.637,153.712
C05150=1087.994,323.244,412.105,176.899,23.633,153.711
C05151=1087.989,322.997,412.138,176.896,23.629,153.711
C05152=1087.983,322.749,412.170,176.893,23.625,153.710
C05153=1087.977,322.501,412.202,176.890,23.622,153.710
C05154=1087.971,322.253,412.236,176.887,23.618,153.709
C05155=1087.966,322.005,412.267,176.883,23.614,153.709
C05156=1087.959,321.758,412.300,176.881,23.610,153.709
C05157=1087.953,321.509,412.332,176.878,23.606,153.708
C05158=1087.949,321.262,412.365,176.875,23.602,153.708
C05159=1087.943,321.014,412.397,176.872,23.598,153.707
C05160=1087.937,320.766,412.429,176.868,23.594,153.707
C05161=1087.930,320.518,412.462,176.866,23.590,153.706
C05162=1087.926,320.270,412.494,176.863,23.586,153.706
C05163=1087.920,320.022,412.526,176.860,23.583,153.705
C05164=1087.914,319.775,412.559,176.857,23.579,153.705
C05165=1087.908,319.527,412.591,176.854,23.575,153.704
C05166=1087.902,319.279,412.623,176.850,23.571,153.704
C05167=1087.897,319.031,412.655,176.848,23.567,153.703
C05168=1087.891,318.783,412.688,176.845,23.563,153.703
C05169=1087.885,318.535,412.720,176.842,23.559,153.702
C05170=1087.880,318.288,412.751,176.839,23.556,153.702
C05171=1087.874,318.039,412.783,176.836,23.552,153.701
C05172=1087.868,317.792,412.815,176.833,23.547,153.701
C05173=1087.863,317.543,412.848,176.830,23.544,153.700
C05174=1087.853,317.140,412.900,176.825,23.538,153.700
C05175=1087.844,316.736,412.952,176.820,23.532,153.699
C05176=1087.835,316.332,413.005,176.815,23.525,153.698
C05177=1087.826,315.930,413.056,176.810,23.519,153.697
C05178=1087.820,315.682,413.088,176.807,23.515,153.697
C05179=1087.815,315.434,413.120,176.804,23.512,153.697
C05180=1087.809,315.186,413.152,176.802,23.508,153.696
C05181=1087.804,314.938,413.184,176.799,23.504,153.696
C05182=1087.797,314.690,413.215,176.796,23.500,153.695
C05183=1087.791,314.442,413.248,176.793,23.497,153.695
C05184=1087.786,314.194,413.279,176.790,23.493,153.694
C05185=1087.780,313.946,413.311,176.786,23.489,153.694
C05186=1087.773,313.698,413.343,176.783,23.485,153.694
C05187=1087.768,313.451,413.374,176.780,23.482,153.693
C05188=1087.762,313.202,413.406,176.777,23.479,153.693
C05189=1087.757,312.954,413.437,176.774,23.475,153.692
C05190=1087.750,312.707,413.469,176.772,23.471,153.692
C05191=1087.745,312.459,413.500,176.769,23.468,153.692
C05192=1087.739,312.211,413.532,176.766,23.464,153.691
C05193=1087.732,311.964,413.563,176.763,23.460,153.691
C05194=1087.727,311.715,413.595,176.759,23.456,153.690
C05195=1087.721,311.467,413.627,176.756,23.453,153.690
C05196=1087.715,311.219,413.658,176.753,23.450,153.690
C05197=1087.709,310.971,413.690,176.750,23.446,153.689
C05198=1087.703,310.724,413.722,176.747,23.442,153.689
C05199=1087.698,310.475,413.753,176.744,23.439,153.688
C05200=1087.692,310.228,413.784,176.742,23.435,153.688
C05201=1087.686,309.980,413.816,176.739,23.431,153.687
C05202=1087.680,309.731,413.847,176.736,23.428,153.687
C05203=1087.674,309.484,413.878,176.733,23.425,153.687
C05204=1087.668,309.236,413.910,176.730,23.421,153.686
C05205=1087.663,308.988,413.941,176.726,23.417,153.686
C05206=1087.657,308.740,413.972,176.723,23.413,153.685
C05207=1087.651,308.492,414.004,176.720,23.410,153.685
C05208=1087.645,308.244,414.034,176.717,23.407,153.685
C05209=1087.639,307.996,414.066,176.714,23.403,153.684
C05210=1087.634,307.748,414.097,176.711,23.399,153.684
C05211=1087.628,307.500,414.129,176.709,23.396,153.683
C05212=1087.622,307.252,414.160,176.706,23.392,153.683
C05213=1087.616,307.005,414.191,176.703,23.389,153.683
C05214=1087.611,306.756,414.222,176.700,23.385,153.682
C05215=1087.605,306.509,414.254,176.697,23.382,153.682
C05216=1087.599,306.261,414.284,176.694,23.378,153.681
C05217=1087.593,306.013,414.316,176.691,23.374,153.681
C05218=1087.588,305.765,414.347,176.688,23.371,153.681
C05219=1087.582,305.517,414.378,176.684,23.367,153.680
C05220=1087.576,305.269,414.409,176.681,23.363,153.680
C05221=1087.570,305.021,414.441,176.678,23.360,153.680
C05222=1087.565,304.773,414.471,176.675,23.357,153.679
C05223=1087.560,304.525,414.502,176.672,23.353,153.679
C05224=1087.554,304.277,414.534,176.670,23.349,153.678
C05225=1087.548,304.029,414.564,176.667,23.346,153.678
C05226=1087.539,303.628,414.614,176.662,23.340,153.677
C05227=1087.530,303.228,414.664,176.657,23.334,153.677
C05228=1087.521,302.827,414.714,176.653,23.329,153.676
C05229=1087.511,302.426,414.764,176.648,23.323,153.675
C05230=1087.505,302.178,414.796,176.645,23.320,153.675
C05231=1087.500,301.930,414.826,176.642,23.316,153.675
C05232=1087.495,301.682,414.857,176.639,23.313,153.674
C05233=1087.489,301.434,414.887,176.636,23.309,153.674
C05234=1087.484,301.186,414.918,176.633,23.306,153.674
C05235=1087.477,300.937,414.949,176.630,23.302,153.673
C05236=1087.471,300.690,414.980,176.627,23.299,153.673
C05237=1087.466,300.442,415.011,176.624,23.295,153.672
C05238=1087.460,300.194,415.041,176.621,23.292,153.672
C05239=1087.455,299.946,415.072,176.618,23.288,153.672
C05240=1087.449,299.698,415.103,176.615,23.285,153.671
C05241=1087.444,299.450,415.134,176.612,23.281,153.671
C05242=1087.438,299.202,415.164,176.610,23.277,153.671
C05243=1087.432,298.954,415.195,176.606,23.274,153.670
C05244=1087.427,298.706,415.226,176.604,23.271,153.670
C05245=1087.421,298.458,415.256,176.601,23.267,153.669
C05246=1087.416,298.210,415.287,176.598,23.264,153.669
C05247=1087.410,297.962,415.317,176.595,23.260,153.669
C05248=1087.404,297.714,415.348,176.592,23.257,153.668
C05249=1087.399,297.466,415.378,176.589,23.253,153.668
C05250=1087.393,297.217,415.409,176.586,23.250,153.668
C05251=1087.387,296.970,415.440,176.583,23.247,153.667
C05252=1087.381,296.722,415.470,176.580,23.243,153.667
C05253=1087.375,296.474,415.500,176.577,23.240,153.667
C05254=1087.370,296.226,415.531,176.574,23.237,153.666
C05255=1087.365,295.977,415.561,176.571,23.233,153.666
C05256=1087.359,295.730,415.591,176.568,23.230,153.666
C05257=1087.353,295.482,415.622,176.565,23.227,153.665
C05258=1087.347,295.233,415.652,176.562,23.223,153.665
C05259=1087.341,294.985,415.683,176.559,23.220,153.665
C05260=1087.335,294.737,415.712,176.556,23.217,153.664
C05261=1087.330,294.489,415.743,176.553,23.213,153.664
C05262=1087.324,294.241,415.773,176.550,23.210,153.664
C05263=1087.318,293.993,415.803,176.547,23.206,153.663
C05264=1087.312,293.745,415.833,176.544,23.203,153.663
C05265=1087.307,293.497,415.863,176.541,23.200,153.663
C05266=1087.302,293.249,415.894,176.538,23.196,153.662
C05267=1087.296,293.001,415.924,176.536,23.193,153.662
C05268=1087.290,292.753,415.954,176.533,23.190,153.662
C05269=1087.284,292.505,415.985,176.530,23.186,153.661
C05270=1087.279,292.257,416.014,176.527,23.183,153.661
C05271=1087.273,292.009,416.045,176.524,23.180,153.660
C05272=1087.267,291.761,416.075,176.521,23.176,153.660
C05273=1087.262,291.512,416.105,176.518,23.173,153.660
C05274=1087.255,291.264,416.135,176.515,23.170,153.659
C05275=1087.250,291.015,416.165,176.512,23.166,153.659
C05276=1087.244,290.768,416.195,176.509,23.163,153.659
C05277=1087.239,290.519,416.225,176.506,23.160,153.659
C05278=1087.230,290.133,416.272,176.502,23.155,153.658
C05279=1087.220,289.746,416.318,176.498,23.150,153.657
C05280=1087.211,289.360,416.365,176.493,23.145,153.657
C05281=1087.203,288.973,416.411,176.489,23.140,153.656
C05282=1087.197,288.726,416.441,176.486,23.136,153.656
C05283=1087.191,288.477,416.471,176.483,23.133,153.656
C05284=1087.186,288.229,416.500,176.480,23.130,153.656
C05285=1087.180,287.981,416.531,176.477,23.126,153.655
C05286=1087.174,287.732,416.560,176.474,23.123,153.655
C05287=1087.168,287.484,416.590,176.471,23.120,153.655
C05288=1087.162,287.236,416.620,176.468,23.117,153.654
C05289=1087.157,286.988,416.649,176.465,23.114,153.654
C05290=1087.151,286.740,416.679,176.462,23.111,153.654
C05291=1087.145,286.492,416.709,176.460,23.107,153.653
C05292=1087.139,286.244,416.739,176.456,23.104,153.653
C05293=1087.134,285.995,416.768,176.453,23.101,153.653
C05294=1087.128,285.747,416.798,176.450,23.098,153.652
C05295=1087.122,285.499,416.828,176.447,23.094,153.652
C05296=1087.117,285.251,416.857,176.445,23.091,153.652
C05297=1087.111,285.003,416.886,176.441,23.088,153.651
C05298=1087.106,284.784,416.913,176.439,23.085,153.651
C05299=1087.101,284.566,416.938,176.437,23.083,153.651
C05300=1087.096,284.348,416.964,176.434,23.079,153.651
C05301=1087.091,284.129,416.990,176.432,23.077,153.650
C05302=1087.086,283.911,417.016,176.429,23.073,153.650
C05303=1087.081,283.692,417.042,176.427,23.071,153.650
C05304=1087.076,283.474,417.069,176.423,23.068,153.650
C05305=1087.071,283.256,417.095,176.421,23.065,153.649
C05306=1087.065,283.008,417.124,176.418,23.062,153.649
C05307=1087.059,282.759,417.153,176.415,23.059,153.649
C05308=1087.054,282.511,417.183,176.412,23.056,153.648
C05309=1087.048,282.263,417.212,176.410,23.052,153.648
C05310=1087.043,282.015,417.241,176.407,23.049,153.648
C05311=1087.037,281.766,417.271,176.404,23.046,153.647
C05312=1087.031,281.518,417.300,176.401,23.043,153.647
C05313=1087.025,281.270,417.330,176.398,23.040,153.647
C05314=1087.020,281.022,417.359,176.395,23.036,153.647
C05315=1087.014,280.774,417.388,176.392,23.033,153.646
C05316=1087.009,280.526,417.418,176.390,23.030,153.646
C05317=1087.002,280.277,417.447,176.387,23.027,153.646
C05318=1086.997,280.029,417.476,176.384,23.024,153.645
C05319=1086.991,279.780,417.505,176.381,23.021,153.645
C05320=1086.986,279.532,417.534,176.378,23.017,153.645
C05321=1086.980,279.284,417.563,176.375,23.014,153.644
C05322=1086.974,279.036,417.593,176.372,23.011,153.644
C05323=1086.968,278.788,417.622,176.370,23.008,153.644
C05324=1086.963,278.540,417.651,176.367,23.005,153.644
C05325=1086.957,278.291,417.679,176.364,23.002,153.643
C05326=1086.952,278.043,417.709,176.361,22.998,153.643
C05327=1086.945,277.795,417.738,176.358,22.995,153.643
C05328=1086.941,277.547,417.767,176.355,22.992,153.642
C05329=1086.934,277.299,417.796,176.353,22.989,153.642
C05330=1086.929,277.080,417.821,176.349,22.987,153.642
C05331=1086.924,276.861,417.847,176.347,22.984,153.642
C05332=1086.919,276.644,417.872,176.345,22.981,153.641
C05333=1086.915,276.425,417.898,176.342,22.978,153.641
C05334=1086.909,276.206,417.923,176.340,22.976,153.641
C05335=1086.904,275.988,417.949,176.337,22.972,153.641
C05336=1086.900,275.770,417.974,176.334,22.970,153.640
C05337=1086.894,275.552,418.000,176.332,22.967,153.640
C05338=1086.888,275.303,418.028,176.329,22.964,153.640
C05339=1086.883,275.056,418.057,176.326,22.961,153.640
C05340=1086.877,274.807,418.086,176.323,22.958,153.639
C05341=1086.872,274.558,418.115,176.320,22.955,153.639
C05342=1086.866,274.311,418.144,176.318,22.952,153.639
C05343=1086.860,274.062,418.172,176.315,22.949,153.638
C05344=1086.855,273.814,418.202,176.312,22.945,153.638
C05345=1086.849,273.566,418.230,176.309,22.942,153.638
C05346=1086.843,273.318,418.259,176.306,22.939,153.638
C05347=1086.837,273.069,418.287,176.304,22.937,153.637
C05348=1086.832,272.821,418.317,176.301,22.934,153.637
C05349=1086.826,272.572,418.345,176.298,22.930,153.637
C05350=1086.820,272.324,418.374,176.295,22.927,153.637
C05351=1086.815,272.076,418.402,176.292,22.924,153.636
C05352=1086.809,271.828,418.432,176.290,22.921,153.636
C05353=1086.804,271.580,418.460,176.287,22.918,153.636
C05354=1086.798,271.331,418.488,176.284,22.915,153.635
C05355=1086.792,271.083,418.517,176.281,22.912,153.635
C05356=1086.786,270.835,418.545,176.278,22.909,153.635
C05357=1086.780,270.587,418.574,176.275,22.906,153.635
C05358=1086.775,270.338,418.603,176.272,22.903,153.634
C05359=1086.770,270.089,418.631,176.269,22.900,153.634
C05360=1086.763,269.841,418.660,176.266,22.896,153.634
C05361=1086.758,269.593,418.688,176.264,22.894,153.634
C05362=1086.752,269.345,418.716,176.261,22.890,153.633
C05363=1086.746,269.097,418.745,176.258,22.887,153.633
C05364=1086.740,268.848,418.773,176.255,22.885,153.633
C05365=1086.735,268.600,418.801,176.253,22.882,153.633
C05366=1086.730,268.351,418.830,176.250,22.879,153.632
C05367=1086.724,268.103,418.859,176.247,22.875,153.632
C05368=1086.718,267.855,418.887,176.244,22.872,153.632
C05369=1086.712,267.606,418.915,176.241,22.869,153.631
C05370=1086.707,267.358,418.943,176.238,22.867,153.631
C05371=1086.701,267.110,418.972,176.235,22.863,153.631
C05372=1086.696,266.861,419.000,176.232,22.860,153.631
C05373=1086.690,266.613,419.029,176.229,22.857,153.630
C05374=1086.684,266.365,419.057,176.227,22.854,153.630
C05375=1086.678,266.117,419.085,176.224,22.851,153.630
C05376=1086.673,265.868,419.113,176.221,22.848,153.630
C05377=1086.667,265.620,419.141,176.218,22.845,153.629
C05378=1086.662,265.372,419.169,176.216,22.842,153.629
C05379=1086.656,265.123,419.198,176.213,22.839,153.629
C05380=1086.650,264.875,419.225,176.210,22.836,153.629
C05381=1086.644,264.626,419.254,176.207,22.833,153.628
C05382=1086.639,264.378,419.282,176.205,22.830,153.628
C05383=1086.633,264.129,419.310,176.202,22.827,153.628
C05384=1086.628,263.881,419.338,176.199,22.824,153.628
C05385=1086.621,263.633,419.366,176.196,22.822,153.627
C05386=1086.613,263.259,419.408,176.192,22.817,153.627
C05387=1086.604,262.884,419.450,176.187,22.813,153.627
C05388=1086.595,262.510,419.493,176.183,22.808,153.626
C05389=1086.586,262.136,419.534,176.179,22.804,153.626
C05390=1086.580,261.887,419.562,176.176,22.801,153.626
C05391=1086.575,261.639,419.590,176.174,22.798,153.625
C05392=1086.569,261.390,419.619,176.170,22.795,153.625
C05393=1086.563,261.142,419.645,176.167,22.792,153.625
C05394=1086.557,260.893,419.674,176.164,22.789,153.625
C05395=1086.552,260.645,419.702,176.162,22.786,153.625
C05396=1086.545,260.397,419.729,176.159,22.783,153.624
C05397=1086.540,260.149,419.757,176.156,22.780,153.624
C05398=1086.535,259.900,419.785,176.154,22.778,153.624
C05399=1086.529,259.651,419.813,176.151,22.774,153.624
C05400=1086.523,259.404,419.840,176.148,22.771,153.623
C05401=1086.517,259.155,419.869,176.145,22.768,153.623
C05402=1086.512,258.906,419.896,176.142,22.766,153.623
C05403=1086.506,258.659,419.923,176.139,22.762,153.623
C05404=1086.500,258.410,419.952,176.136,22.760,153.622
C05405=1086.495,258.161,419.979,176.134,22.757,153.622
C05406=1086.488,257.913,420.007,176.131,22.754,153.622
C05407=1086.483,257.665,420.035,176.128,22.751,153.622
C05408=1086.477,257.416,420.061,176.126,22.748,153.621
C05409=1086.471,257.167,420.089,176.123,22.745,153.621
C05410=1086.466,256.919,420.117,176.120,22.742,153.621
C05411=1086.460,256.671,420.144,176.117,22.739,153.621
C05412=1086.454,256.422,420.172,176.115,22.736,153.620
C05413=1086.449,256.174,420.200,176.112,22.733,153.620
C05414=1086.443,255.926,420.227,176.108,22.730,153.620
C05415=1086.437,255.677,420.255,176.106,22.728,153.620
C05416=1086.431,255.429,420.282,176.103,22.724,153.619
C05417=1086.426,255.180,420.309,176.100,22.722,153.619
C05418=1086.421,254.932,420.337,176.098,22.719,153.619
C05419=1086.414,254.683,420.364,176.095,22.716,153.619
C05420=1086.409,254.435,420.392,176.092,22.713,153.619
C05421=1086.403,254.187,420.419,176.090,22.710,153.618
C05422=1086.397,253.938,420.447,176.087,22.707,153.618
C05423=1086.392,253.689,420.474,176.084,22.704,153.618
C05424=1086.386,253.441,420.502,176.081,22.701,153.617
C05425=1086.381,253.193,420.529,176.078,22.698,153.617
C05426=1086.375,252.944,420.556,176.075,22.695,153.617
C05427=1086.369,252.696,420.584,176.073,22.693,153.617
C05428=1086.364,252.447,420.611,176.070,22.689,153.617
C05429=1086.359,252.199,420.638,176.067,22.686,153.616
C05430=1086.353,251.951,420.665,176.065,22.684,153.616
C05431=1086.347,251.701,420.693,176.062,22.681,153.616
C05432=1086.341,251.453,420.719,176.059,22.677,153.616
C05433=1086.336,251.205,420.747,176.057,22.675,153.615
C05434=1086.330,250.957,420.774,176.054,22.672,153.615
C05435=1086.325,250.708,420.801,176.051,22.669,153.615
C05436=1086.319,250.460,420.829,176.048,22.666,153.614
C05437=1086.313,250.211,420.856,176.045,22.663,153.614
C05438=1086.305,249.834,420.897,176.042,22.659,153.614
C05439=1086.297,249.457,420.939,176.037,22.654,153.614
C05440=1086.288,249.080,420.979,176.033,22.649,153.613
C05441=1086.280,248.702,421.020,176.029,22.645,153.613
C05442=1086.275,248.454,421.047,176.026,22.642,153.613
C05443=1086.269,248.206,421.075,176.024,22.639,153.612
C05444=1086.264,247.957,421.102,176.021,22.636,153.612
C05445=1086.258,247.709,421.129,176.018,22.633,153.612
C05446=1086.253,247.460,421.156,176.016,22.630,153.612
C05447=1086.247,247.212,421.183,176.012,22.627,153.611
C05448=1086.241,246.963,421.210,176.009,22.624,153.611
C05449=1086.236,246.714,421.237,176.007,22.621,153.611
C05450=1086.230,246.466,421.264,176.004,22.619,153.611
C05451=1086.224,246.217,421.290,176.002,22.616,153.610
C05452=1086.218,245.969,421.317,175.999,22.613,153.610
C05453=1086.213,245.720,421.344,175.996,22.610,153.610
C05454=1086.207,245.472,421.371,175.994,22.607,153.610
C05455=1086.202,245.224,421.397,175.991,22.604,153.610
C05456=1086.196,244.975,421.424,175.988,22.602,153.609
C05457=1086.191,244.727,421.451,175.985,22.598,153.609
C05458=1086.184,244.478,421.478,175.982,22.596,153.609
